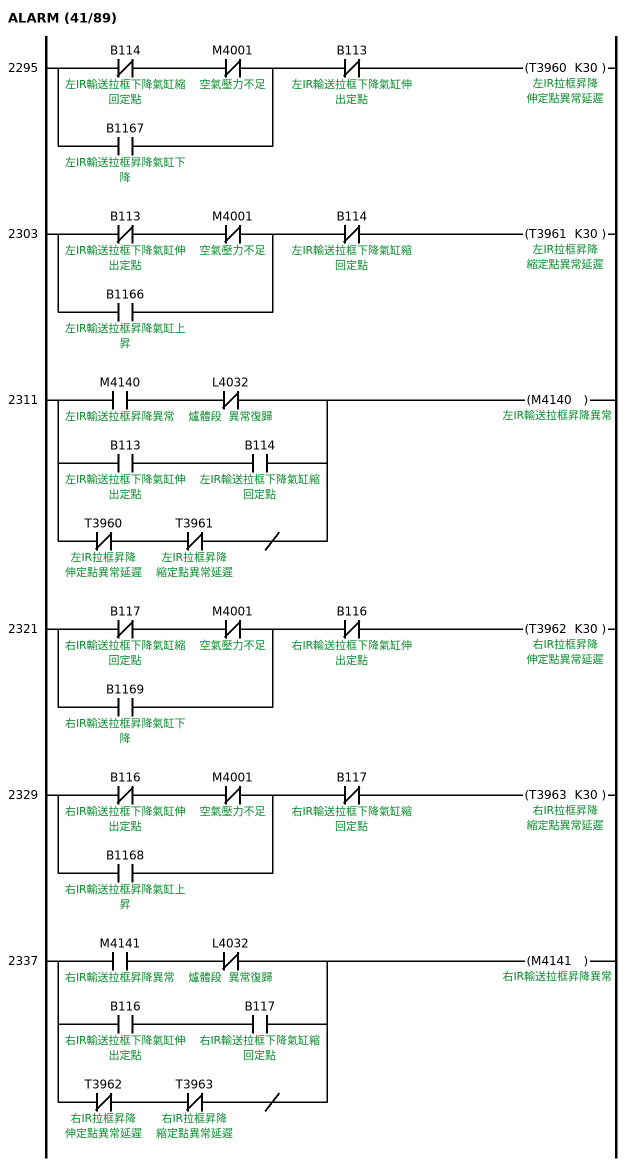
[picture p216: ladder of ALARM, rungs at steps 2295 to 2337]
2295  LDI     B114  ; 左IR輸送拉框下降氣缸縮回定點
      ANI     M4001  ; 空氣壓力不足
      OR      B1167  ; 左IR輸送拉框昇降氣缸下降
      ANI     B113  ; 左IR輸送拉框下降氣缸伸出定點
      OUT     T3960 K30  ; 左IR拉框昇降  伸定點異常延遲
2303  LDI     B113  ; 左IR輸送拉框下降氣缸伸出定點
      ANI     M4001  ; 空氣壓力不足
      OR      B1166  ; 左IR輸送拉框昇降氣缸上昇
      ANI     B114  ; 左IR輸送拉框下降氣缸縮回定點
      OUT     T3961 K30  ; 左IR拉框昇降  縮定點異常延遲
2311  LD      M4140  ; 左IR輸送拉框昇降異常
      ANI     L4032  ; 爐體段  異常復歸
      LD      B113  ; 左IR輸送拉框下降氣缸伸出定點
      AND     B114  ; 左IR輸送拉框下降氣缸縮回定點
      ORB
      LDI     T3960  ; 左IR拉框昇降  伸定點異常延遲
      ANI     T3961  ; 左IR拉框昇降  縮定點異常延遲
      INV
      ORB
      OUT     M4140  ; 左IR輸送拉框昇降異常
2321  LDI     B117  ; 右IR輸送拉框下降氣缸縮回定點
      ANI     M4001  ; 空氣壓力不足
      OR      B1169  ; 右IR輸送拉框昇降氣缸下降
      ANI     B116  ; 右IR輸送拉框下降氣缸伸出定點
      OUT     T3962 K30  ; 右IR拉框昇降  伸定點異常延遲
2329  LDI     B116  ; 右IR輸送拉框下降氣缸伸出定點
      ANI     M4001  ; 空氣壓力不足
      OR      B1168  ; 右IR輸送拉框昇降氣缸上昇
      ANI     B117  ; 右IR輸送拉框下降氣缸縮回定點
      OUT     T3963 K30  ; 右IR拉框昇降  縮定點異常延遲
2337  LD      M4141  ; 右IR輸送拉框昇降異常
      ANI     L4032  ; 爐體段  異常復歸
      LD      B116  ; 右IR輸送拉框下降氣缸伸出定點
      AND     B117  ; 右IR輸送拉框下降氣缸縮回定點
      ORB
      LDI     T3962  ; 右IR拉框昇降  伸定點異常延遲
      ANI     T3963  ; 右IR拉框昇降  縮定點異常延遲
      INV
      ORB
      OUT     M4141  ; 右IR輸送拉框昇降異常
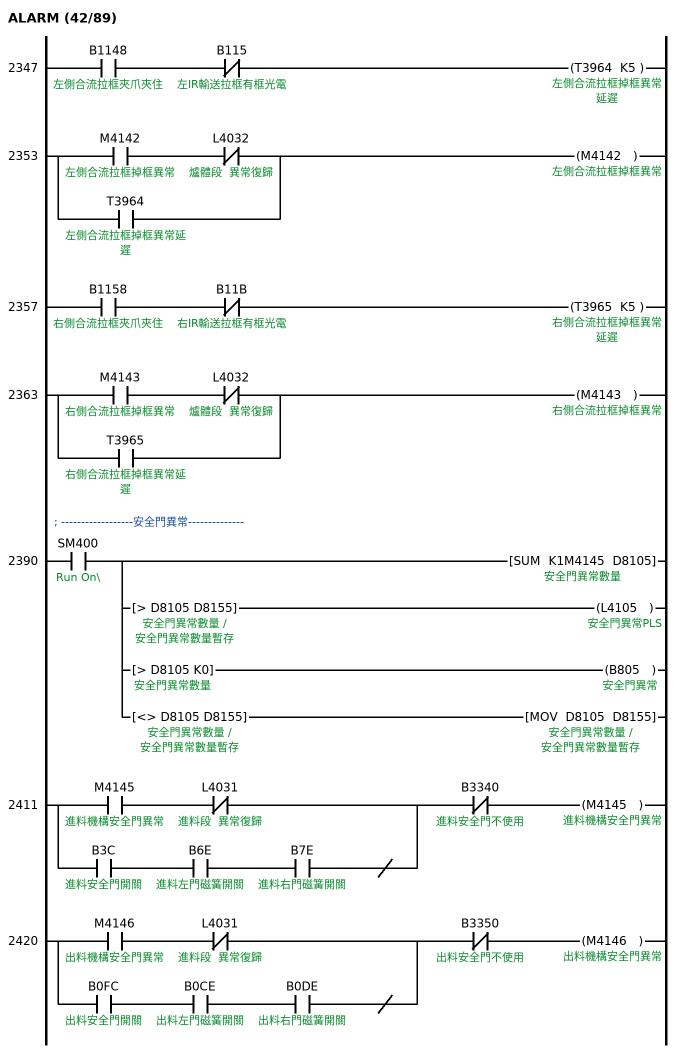
2347  LD      B1148  ; 左側合流拉框夾爪夾住
      ANI     B115  ; 左IR輸送拉框有框光電
      OUT     T3964 K5  ; 左側合流拉框掉框異常延遲
2353  LD      M4142  ; 左側合流拉框掉框異常
      ANI     L4032  ; 爐體段  異常復歸
      OR      T3964  ; 左側合流拉框掉框異常延遲
      OUT     M4142  ; 左側合流拉框掉框異常
2357  LD      B1158  ; 右側合流拉框夾爪夾住
      ANI     B11B  ; 右IR輸送拉框有框光電
      OUT     T3965 K5  ; 右側合流拉框掉框異常延遲
2363  LD      M4143  ; 右側合流拉框掉框異常
      ANI     L4032  ; 爐體段  異常復歸
      OR      T3965  ; 右側合流拉框掉框異常延遲
      OUT     M4143  ; 右側合流拉框掉框異常
; ------------------安全門異常--------------
2390  LD      SM400  ; Run On\
      SUM     K1M4145 D8105  ; 進料機構安全門異常 / 安全門異常數量
      MPS
      AND>    D8105 D8155  ; 安全門異常數量 / 安全門異常數量暫存
      OUT     L4105  ; 安全門異常PLS
      MRD
      AND>    D8105 K0  ; 安全門異常數量
      OUT     B805  ; 安全門異常
      MPP
      AND<>   D8105 D8155  ; 安全門異常數量 / 安全門異常數量暫存
      MOV     D8105 D8155
2411  LD      M4145  ; 進料機構安全門異常
      ANI     L4031  ; 進料段  異常復歸
      LD      B3C  ; 進料安全門開關
      AND     B6E  ; 進料左門磁簧開關
      AND     B7E  ; 進料右門磁簧開關
      INV
      ORB
      ANI     B3340  ; 進料安全門不使用
      OUT     M4145  ; 進料機構安全門異常
2420  LD      M4146  ; 出料機構安全門異常
      ANI     L4031  ; 進料段  異常復歸
      LD      B0FC  ; 出料安全門開關
      AND     B0CE  ; 出料左門磁簧開關
      AND     B0DE  ; 出料右門磁簧開關
      INV
      ORB
      ANI     B3350  ; 出料安全門不使用
      OUT     M4146  ; 出料機構安全門異常
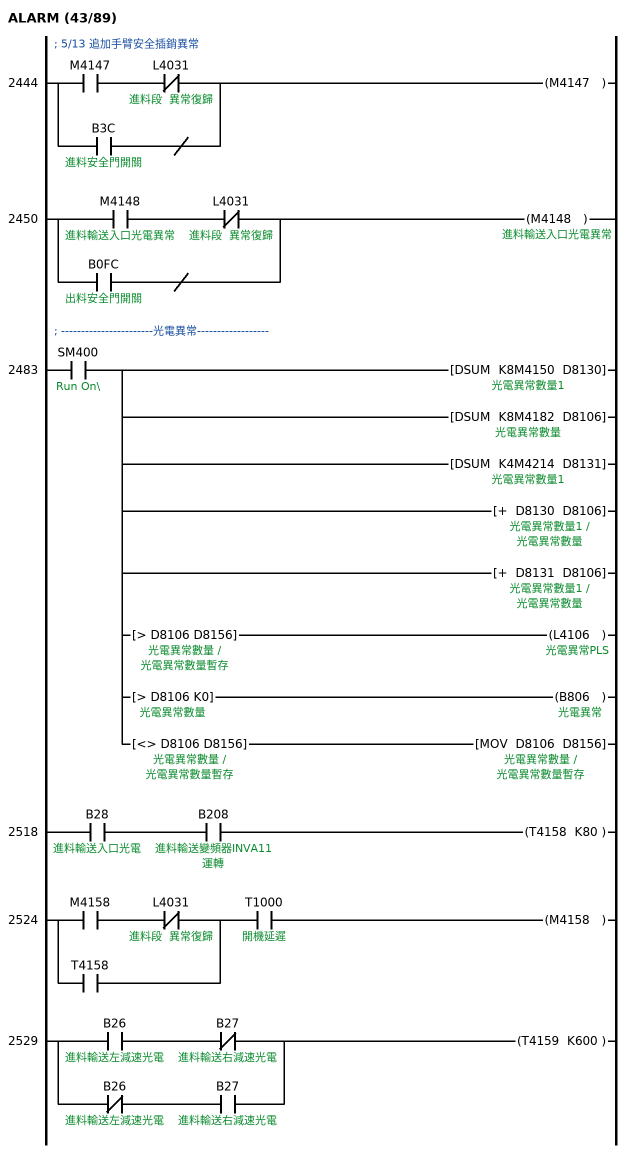
; 5/13 追加手臂安全插銷異常
2444  LD      M4147
      ANI     L4031  ; 進料段  異常復歸
      LD      B3C  ; 進料安全門開關
      INV
      ORB
      OUT     M4147
2450  LD      M4148  ; 進料輸送入口光電異常
      ANI     L4031  ; 進料段  異常復歸
      LD      B0FC  ; 出料安全門開關
      INV
      ORB
      OUT     M4148  ; 進料輸送入口光電異常
; -----------------------光電異常------------------
2483  LD      SM400  ; Run On\
      DSUM    K8M4150 D8130  ; 進料輸送有板光纖異常 / 光電異常數量1
      DSUM    K8M4182 D8106  ; 出料卡板異常 / 光電異常數量
      DSUM    K4M4214 D8131  ; 光電異常數量1
      +       D8130 D8106
      +       D8131 D8106
      MPS
      AND>    D8106 D8156  ; 光電異常數量 / 光電異常數量暫存
      OUT     L4106  ; 光電異常PLS
      MRD
      AND>    D8106 K0  ; 光電異常數量
      OUT     B806  ; 光電異常
      MPP
      AND<>   D8106 D8156  ; 光電異常數量 / 光電異常數量暫存
      MOV     D8106 D8156
2518  LD      B28  ; 進料輸送入口光電
      AND     B208  ; 進料輸送變頻器INVA11運轉
      OUT     T4158 K80
2524  LD      M4158
      ANI     L4031  ; 進料段  異常復歸
      OR      T4158
      AND     T1000  ; 開機延遲
      OUT     M4158
2529  LD      B26  ; 進料輸送左減速光電
      ANI     B27  ; 進料輸送右減速光電
      LDI     B26  ; 進料輸送左減速光電
      AND     B27  ; 進料輸送右減速光電
      ORB
      OUT     T4159 K600
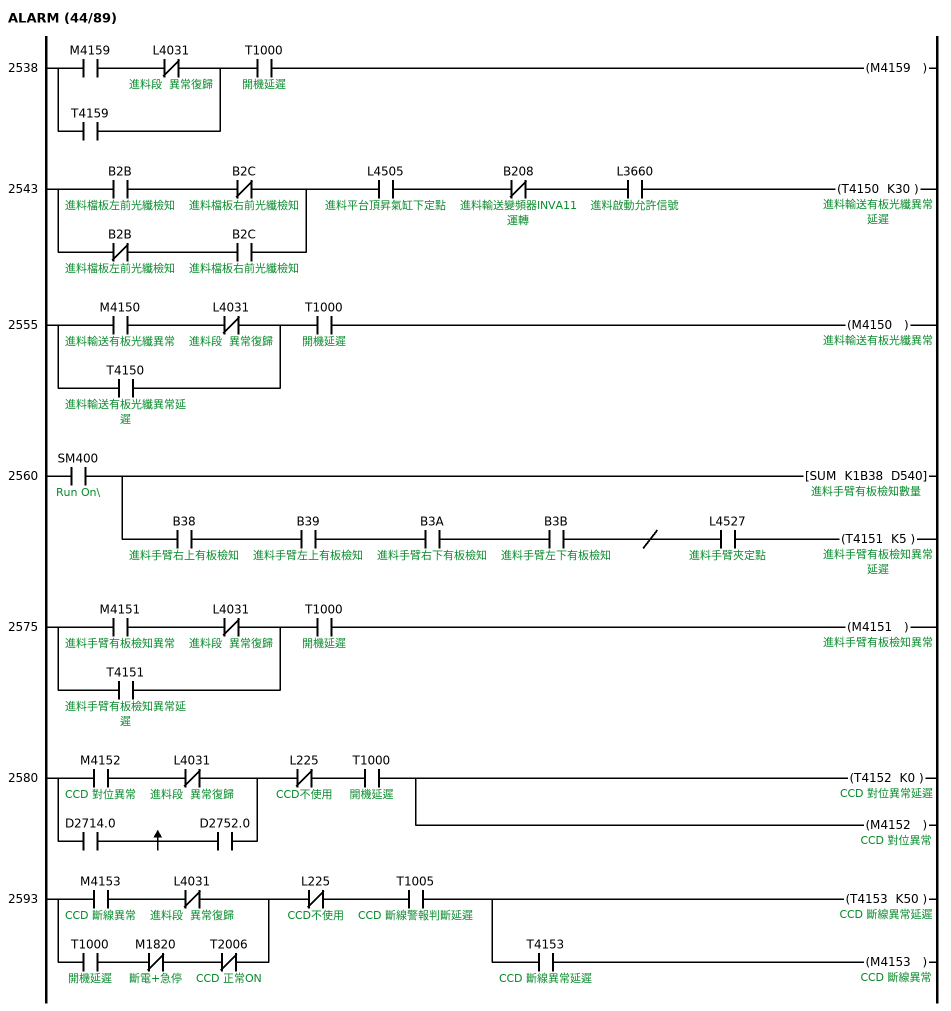
2538  LD      M4159
      ANI     L4031  ; 進料段  異常復歸
      OR      T4159
      AND     T1000  ; 開機延遲
      OUT     M4159
2543  LD      B2B  ; 進料檔板左前光纖檢知
      ANI     B2C  ; 進料檔板右前光纖檢知
      LDI     B2B  ; 進料檔板左前光纖檢知
      AND     B2C  ; 進料檔板右前光纖檢知
      ORB
      AND     L4505  ; 進料平台頂昇氣缸下定點
      ANI     B208  ; 進料輸送變頻器INVA11運轉
      AND     L3660  ; 進料啟動允許信號
      OUT     T4150 K30  ; 進料輸送有板光纖異常延遲
2555  LD      M4150  ; 進料輸送有板光纖異常
      ANI     L4031  ; 進料段  異常復歸
      OR      T4150  ; 進料輸送有板光纖異常延遲
      AND     T1000  ; 開機延遲
      OUT     M4150  ; 進料輸送有板光纖異常
2560  LD      SM400  ; Run On\
      SUM     K1B38 D540  ; 進料手臂右上有板檢知 / 進料手臂有板檢知數量
      AND     B38  ; 進料手臂右上有板檢知
      AND     B39  ; 進料手臂左上有板檢知
      AND     B3A  ; 進料手臂右下有板檢知
      AND     B3B  ; 進料手臂左下有板檢知
      INV
      AND     L4527  ; 進料手臂夾定點
      OUT     T4151 K5  ; 進料手臂有板檢知異常延遲
2575  LD      M4151  ; 進料手臂有板檢知異常
      ANI     L4031  ; 進料段  異常復歸
      OR      T4151  ; 進料手臂有板檢知異常延遲
      AND     T1000  ; 開機延遲
      OUT     M4151  ; 進料手臂有板檢知異常
2580  LD      M4152  ; CCD 對位異常
      ANI     L4031  ; 進料段  異常復歸
      LD      D2714.0
      MEP
      AND     D2752.0
      ORB
      ANI     L225  ; CCD不使用
      AND     T1000  ; 開機延遲
      OUT     T4152 K0  ; CCD 對位異常延遲
      OUT     M4152  ; CCD 對位異常
2593  LD      M4153  ; CCD 斷線異常
      ANI     L4031  ; 進料段  異常復歸
      LD      T1000  ; 開機延遲
      ANI     M1820  ; 斷電+急停
      ANI     T2006  ; CCD 正常ON
      ORB
      ANI     L225  ; CCD不使用
      AND     T1005  ; CCD 斷線警報判斷延遲
      OUT     T4153 K50  ; CCD 斷線異常延遲
      AND     T4153  ; CCD 斷線異常延遲
      OUT     M4153  ; CCD 斷線異常
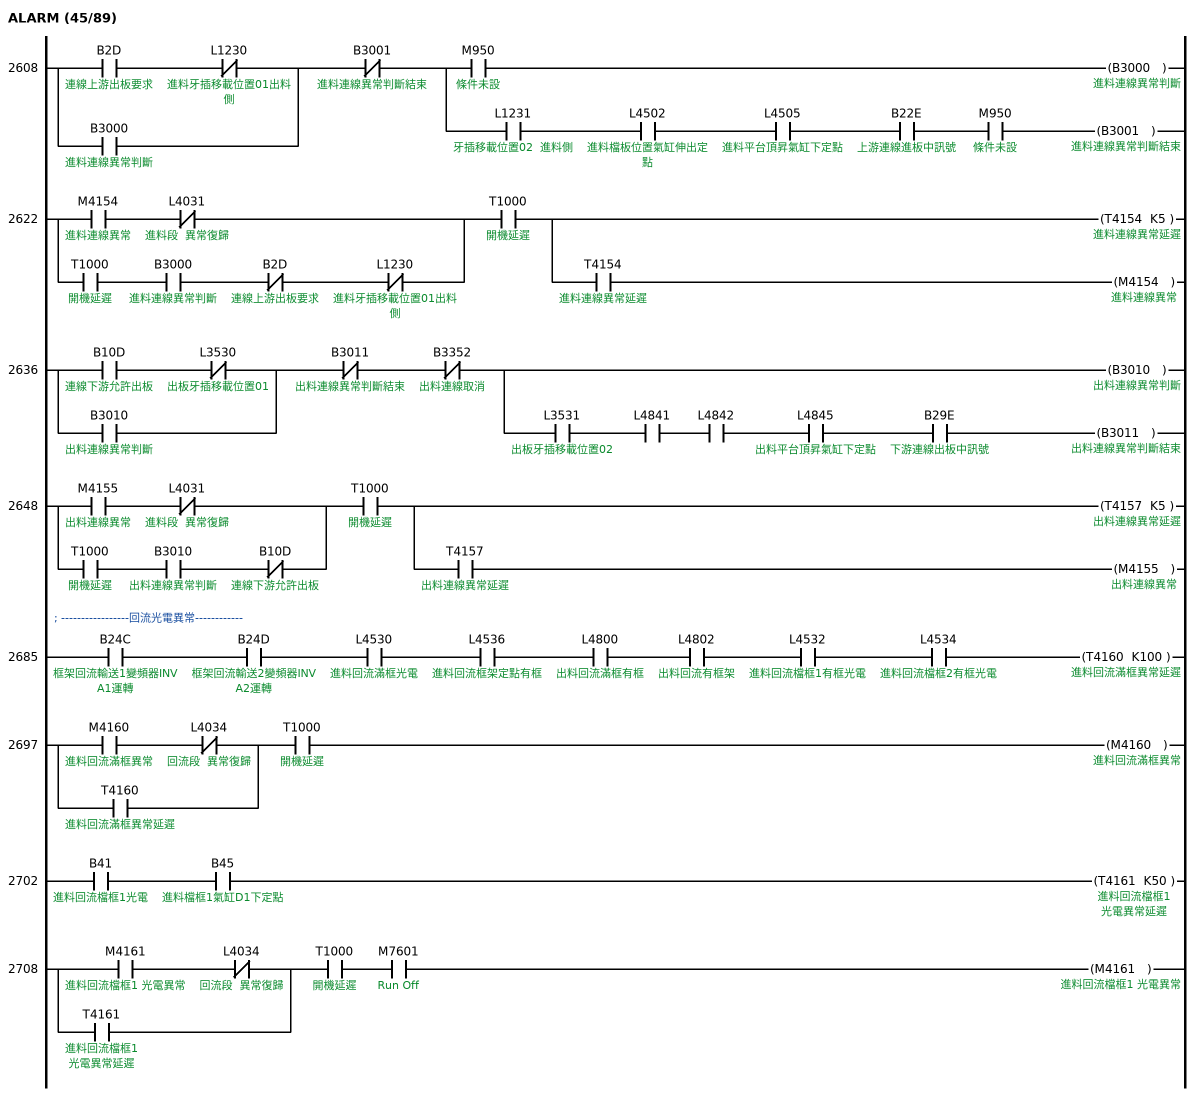
2608  LD      B2D  ; 連線上游出板要求
      ANI     L1230  ; 進料牙插移載位置01出料側
      OR      B3000  ; 進料連線異常判斷
      ANI     B3001  ; 進料連線異常判斷結束
      MPS
      AND     M950  ; 條件未設
      OUT     B3000  ; 進料連線異常判斷
      MPP
      AND     L1231  ; 牙插移載位置02  進料側
      AND     L4502  ; 進料檔板位置氣缸伸出定點
      AND     L4505  ; 進料平台頂昇氣缸下定點
      AND     B22E  ; 上游連線進板中訊號
      AND     M950  ; 條件未設
      OUT     B3001  ; 進料連線異常判斷結束
2622  LD      M4154  ; 進料連線異常
      ANI     L4031  ; 進料段  異常復歸
      LD      T1000  ; 開機延遲
      AND     B3000  ; 進料連線異常判斷
      ANI     B2D  ; 連線上游出板要求
      ANI     L1230  ; 進料牙插移載位置01出料側
      ORB
      AND     T1000  ; 開機延遲
      OUT     T4154 K5  ; 進料連線異常延遲
      AND     T4154  ; 進料連線異常延遲
      OUT     M4154  ; 進料連線異常
2636  LD      B10D  ; 連線下游允許出板
      ANI     L3530  ; 出板牙插移載位置01
      OR      B3010  ; 出料連線異常判斷
      ANI     B3011  ; 出料連線異常判斷結束
      ANI     B3352  ; 出料連線取消
      OUT     B3010  ; 出料連線異常判斷
      AND     L3531  ; 出板牙插移載位置02
      AND     L4841
      AND     L4842
      AND     L4845  ; 出料平台頂昇氣缸下定點
      AND     B29E  ; 下游連線出板中訊號
      OUT     B3011  ; 出料連線異常判斷結束
2648  LD      M4155  ; 出料連線異常
      ANI     L4031  ; 進料段  異常復歸
      LD      T1000  ; 開機延遲
      AND     B3010  ; 出料連線異常判斷
      ANI     B10D  ; 連線下游允許出板
      ORB
      AND     T1000  ; 開機延遲
      OUT     T4157 K5  ; 出料連線異常延遲
      AND     T4157  ; 出料連線異常延遲
      OUT     M4155  ; 出料連線異常
; -----------------回流光電異常------------
2685  LD      B24C  ; 框架回流輸送1變頻器INVA1運轉
      AND     B24D  ; 框架回流輸送2變頻器INVA2運轉
      AND     L4530  ; 進料回流滿框光電
      AND     L4536  ; 進料回流框架定點有框
      AND     L4800  ; 出料回流滿框有框
      AND     L4802  ; 出料回流有框架
      AND     L4532  ; 進料回流檔框1有框光電
      AND     L4534  ; 進料回流檔框2有框光電
      OUT     T4160 K100  ; 進料回流滿框異常延遲
2697  LD      M4160  ; 進料回流滿框異常
      ANI     L4034  ; 回流段  異常復歸
      OR      T4160  ; 進料回流滿框異常延遲
      AND     T1000  ; 開機延遲
      OUT     M4160  ; 進料回流滿框異常
2702  LD      B41  ; 進料回流檔框1光電
      AND     B45  ; 進料檔框1氣缸D1下定點
      OUT     T4161 K50  ; 進料回流檔框1 光電異常延遲
2708  LD      M4161  ; 進料回流檔框1 光電異常
      ANI     L4034  ; 回流段  異常復歸
      OR      T4161  ; 進料回流檔框1 光電異常延遲
      AND     T1000  ; 開機延遲
      AND     M7601  ; Run Off
      OUT     M4161  ; 進料回流檔框1 光電異常
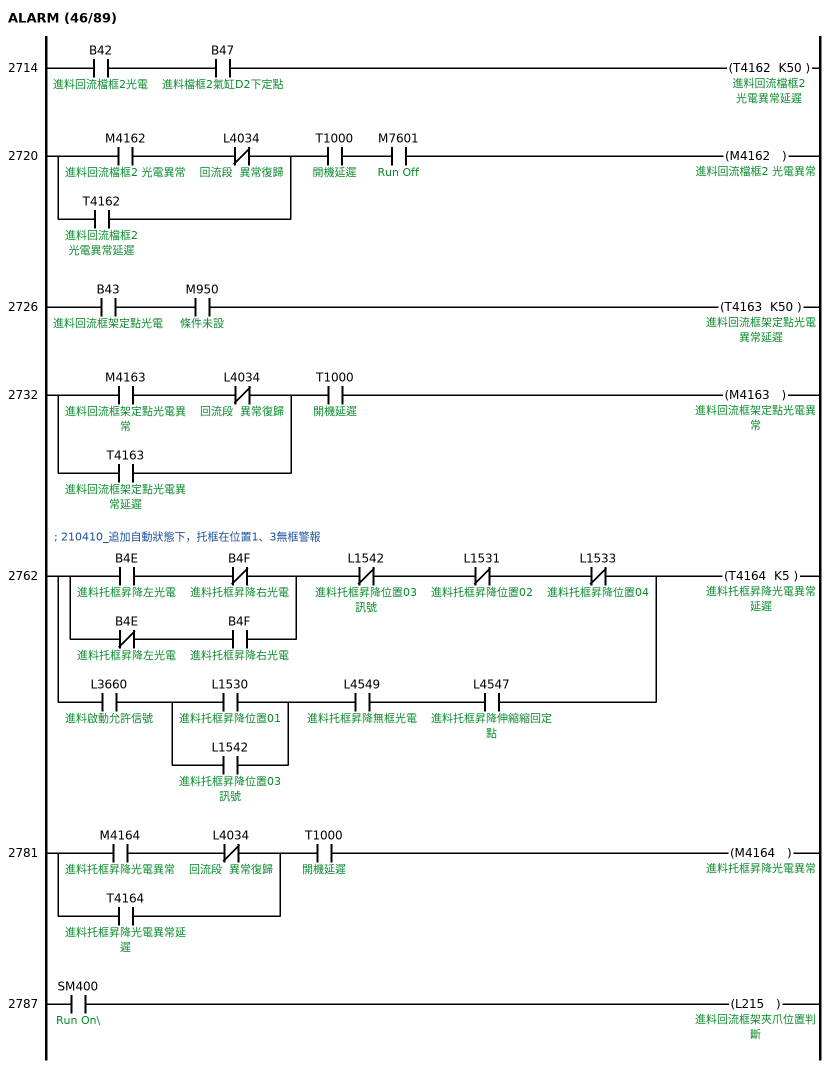
2714  LD      B42  ; 進料回流檔框2光電
      AND     B47  ; 進料檔框2氣缸D2下定點
      OUT     T4162 K50  ; 進料回流檔框2 光電異常延遲
2720  LD      M4162  ; 進料回流檔框2 光電異常
      ANI     L4034  ; 回流段  異常復歸
      OR      T4162  ; 進料回流檔框2 光電異常延遲
      AND     T1000  ; 開機延遲
      AND     M7601  ; Run Off
      OUT     M4162  ; 進料回流檔框2 光電異常
2726  LD      B43  ; 進料回流框架定點光電
      AND     M950  ; 條件未設
      OUT     T4163 K50  ; 進料回流框架定點光電異常延遲
2732  LD      M4163  ; 進料回流框架定點光電異常
      ANI     L4034  ; 回流段  異常復歸
      OR      T4163  ; 進料回流框架定點光電異常延遲
      AND     T1000  ; 開機延遲
      OUT     M4163  ; 進料回流框架定點光電異常
; 210410_追加自動狀態下，托框在位置1、3無框警報
2762  LD      B4E  ; 進料托框昇降左光電
      ANI     B4F  ; 進料托框昇降右光電
      LDI     B4E  ; 進料托框昇降左光電
      AND     B4F  ; 進料托框昇降右光電
      ORB
      ANI     L1542  ; 進料托框昇降位置03 訊號
      ANI     L1531  ; 進料托框昇降位置02
      ANI     L1533  ; 進料托框昇降位置04
      LD      L3660  ; 進料啟動允許信號
      LD      L1530  ; 進料托框昇降位置01
      OR      L1542  ; 進料托框昇降位置03 訊號
      ANB
      AND     L4549  ; 進料托框昇降無框光電
      AND     L4547  ; 進料托框昇降伸縮縮回定點
      ORB
      OUT     T4164 K5  ; 進料托框昇降光電異常延遲
2781  LD      M4164  ; 進料托框昇降光電異常
      ANI     L4034  ; 回流段  異常復歸
      OR      T4164  ; 進料托框昇降光電異常延遲
      AND     T1000  ; 開機延遲
      OUT     M4164  ; 進料托框昇降光電異常
2787  LD      SM400  ; Run On\
      OUT     L215  ; 進料回流框架夾爪位置判斷
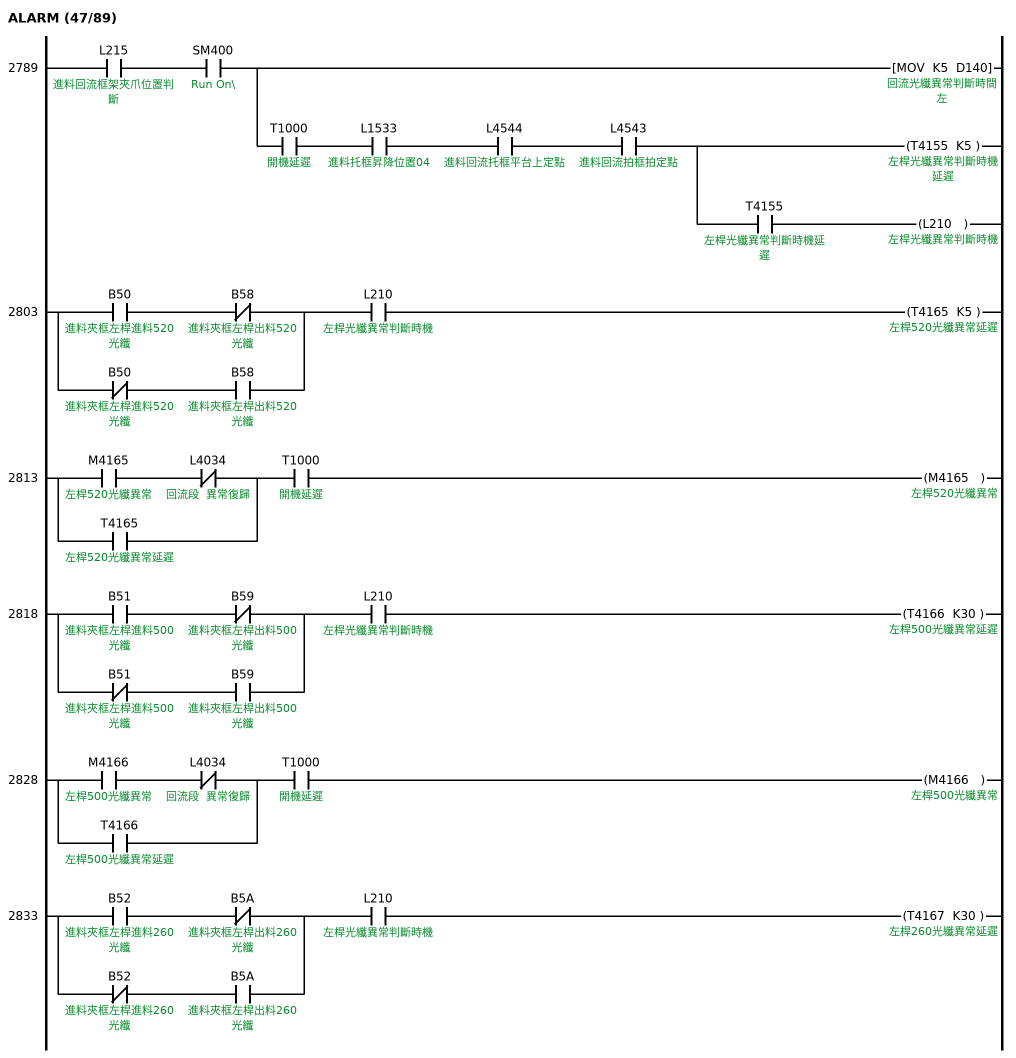
2789  LD      L215  ; 進料回流框架夾爪位置判斷
      AND     SM400  ; Run On\
      MOV     K5 D140  ; 回流光纖異常判斷時間左
      AND     T1000  ; 開機延遲
      AND     L1533  ; 進料托框昇降位置04
      AND     L4544  ; 進料回流托框平台上定點
      AND     L4543  ; 進料回流拍框拍定點
      OUT     T4155 K5  ; 左桿光纖異常判斷時機延遲
      AND     T4155  ; 左桿光纖異常判斷時機延遲
      OUT     L210  ; 左桿光纖異常判斷時機
2803  LD      B50  ; 進料夾框左桿進料520 光纖
      ANI     B58  ; 進料夾框左桿出料520 光纖
      LDI     B50  ; 進料夾框左桿進料520 光纖
      AND     B58  ; 進料夾框左桿出料520 光纖
      ORB
      AND     L210  ; 左桿光纖異常判斷時機
      OUT     T4165 K5  ; 左桿520光纖異常延遲
2813  LD      M4165  ; 左桿520光纖異常
      ANI     L4034  ; 回流段  異常復歸
      OR      T4165  ; 左桿520光纖異常延遲
      AND     T1000  ; 開機延遲
      OUT     M4165  ; 左桿520光纖異常
2818  LD      B51  ; 進料夾框左桿進料500 光纖
      ANI     B59  ; 進料夾框左桿出料500 光纖
      LDI     B51  ; 進料夾框左桿進料500 光纖
      AND     B59  ; 進料夾框左桿出料500 光纖
      ORB
      AND     L210  ; 左桿光纖異常判斷時機
      OUT     T4166 K30  ; 左桿500光纖異常延遲
2828  LD      M4166  ; 左桿500光纖異常
      ANI     L4034  ; 回流段  異常復歸
      OR      T4166  ; 左桿500光纖異常延遲
      AND     T1000  ; 開機延遲
      OUT     M4166  ; 左桿500光纖異常
2833  LD      B52  ; 進料夾框左桿進料260 光纖
      ANI     B5A  ; 進料夾框左桿出料260 光纖
      LDI     B52  ; 進料夾框左桿進料260 光纖
      AND     B5A  ; 進料夾框左桿出料260 光纖
      ORB
      AND     L210  ; 左桿光纖異常判斷時機
      OUT     T4167 K30  ; 左桿260光纖異常延遲
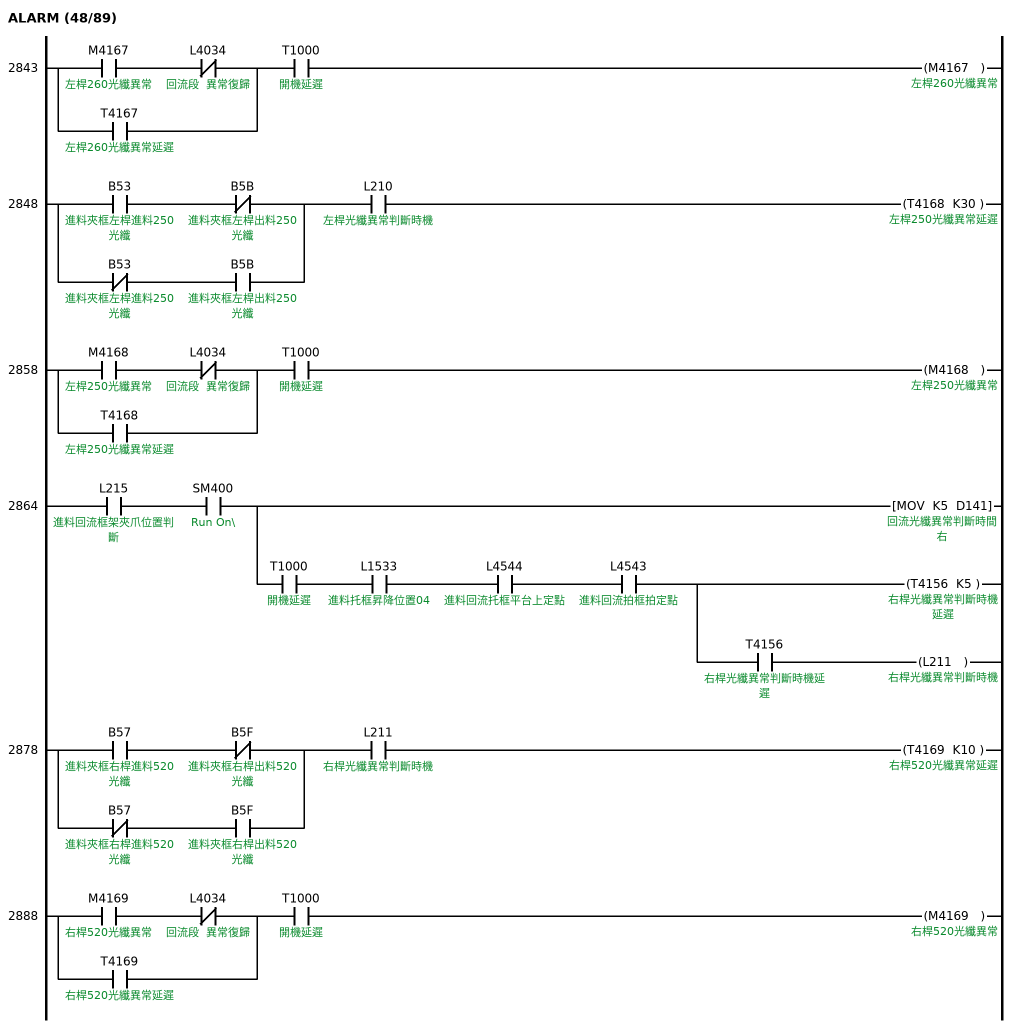
2843  LD      M4167  ; 左桿260光纖異常
      ANI     L4034  ; 回流段  異常復歸
      OR      T4167  ; 左桿260光纖異常延遲
      AND     T1000  ; 開機延遲
      OUT     M4167  ; 左桿260光纖異常
2848  LD      B53  ; 進料夾框左桿進料250 光纖
      ANI     B5B  ; 進料夾框左桿出料250 光纖
      LDI     B53  ; 進料夾框左桿進料250 光纖
      AND     B5B  ; 進料夾框左桿出料250 光纖
      ORB
      AND     L210  ; 左桿光纖異常判斷時機
      OUT     T4168 K30  ; 左桿250光纖異常延遲
2858  LD      M4168  ; 左桿250光纖異常
      ANI     L4034  ; 回流段  異常復歸
      OR      T4168  ; 左桿250光纖異常延遲
      AND     T1000  ; 開機延遲
      OUT     M4168  ; 左桿250光纖異常
2864  LD      L215  ; 進料回流框架夾爪位置判斷
      AND     SM400  ; Run On\
      MOV     K5 D141  ; 回流光纖異常判斷時間右
      AND     T1000  ; 開機延遲
      AND     L1533  ; 進料托框昇降位置04
      AND     L4544  ; 進料回流托框平台上定點
      AND     L4543  ; 進料回流拍框拍定點
      OUT     T4156 K5  ; 右桿光纖異常判斷時機延遲
      AND     T4156  ; 右桿光纖異常判斷時機延遲
      OUT     L211  ; 右桿光纖異常判斷時機
2878  LD      B57  ; 進料夾框右桿進料520 光纖
      ANI     B5F  ; 進料夾框右桿出料520 光纖
      LDI     B57  ; 進料夾框右桿進料520 光纖
      AND     B5F  ; 進料夾框右桿出料520 光纖
      ORB
      AND     L211  ; 右桿光纖異常判斷時機
      OUT     T4169 K10  ; 右桿520光纖異常延遲
2888  LD      M4169  ; 右桿520光纖異常
      ANI     L4034  ; 回流段  異常復歸
      OR      T4169  ; 右桿520光纖異常延遲
      AND     T1000  ; 開機延遲
      OUT     M4169  ; 右桿520光纖異常
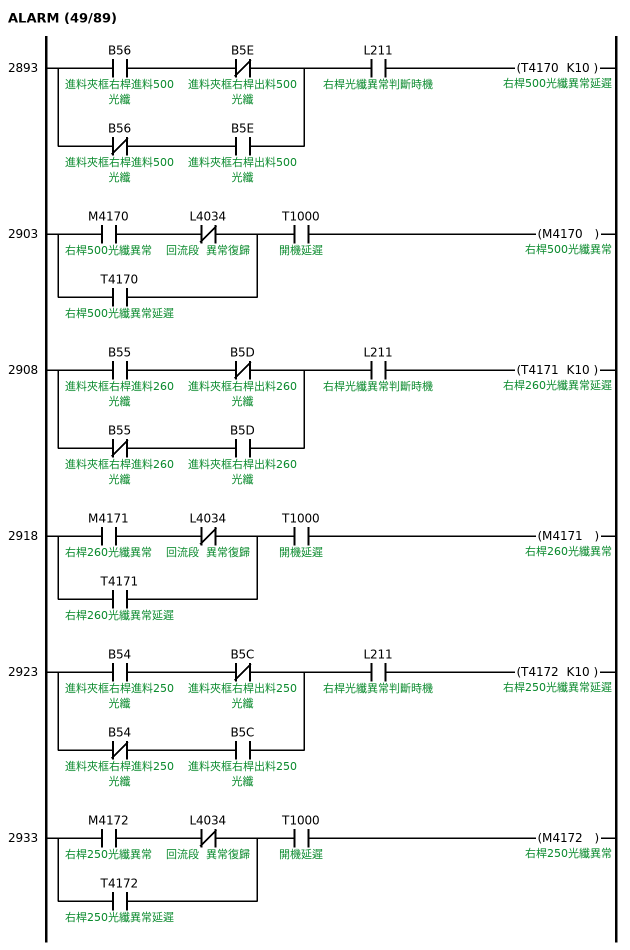
2893  LD      B56  ; 進料夾框右桿進料500 光纖
      ANI     B5E  ; 進料夾框右桿出料500 光纖
      LDI     B56  ; 進料夾框右桿進料500 光纖
      AND     B5E  ; 進料夾框右桿出料500 光纖
      ORB
      AND     L211  ; 右桿光纖異常判斷時機
      OUT     T4170 K10  ; 右桿500光纖異常延遲
2903  LD      M4170  ; 右桿500光纖異常
      ANI     L4034  ; 回流段  異常復歸
      OR      T4170  ; 右桿500光纖異常延遲
      AND     T1000  ; 開機延遲
      OUT     M4170  ; 右桿500光纖異常
2908  LD      B55  ; 進料夾框右桿進料260 光纖
      ANI     B5D  ; 進料夾框右桿出料260 光纖
      LDI     B55  ; 進料夾框右桿進料260 光纖
      AND     B5D  ; 進料夾框右桿出料260 光纖
      ORB
      AND     L211  ; 右桿光纖異常判斷時機
      OUT     T4171 K10  ; 右桿260光纖異常延遲
2918  LD      M4171  ; 右桿260光纖異常
      ANI     L4034  ; 回流段  異常復歸
      OR      T4171  ; 右桿260光纖異常延遲
      AND     T1000  ; 開機延遲
      OUT     M4171  ; 右桿260光纖異常
2923  LD      B54  ; 進料夾框右桿進料250 光纖
      ANI     B5C  ; 進料夾框右桿出料250 光纖
      LDI     B54  ; 進料夾框右桿進料250 光纖
      AND     B5C  ; 進料夾框右桿出料250 光纖
      ORB
      AND     L211  ; 右桿光纖異常判斷時機
      OUT     T4172 K10  ; 右桿250光纖異常延遲
2933  LD      M4172  ; 右桿250光纖異常
      ANI     L4034  ; 回流段  異常復歸
      OR      T4172  ; 右桿250光纖異常延遲
      AND     T1000  ; 開機延遲
      OUT     M4172  ; 右桿250光纖異常
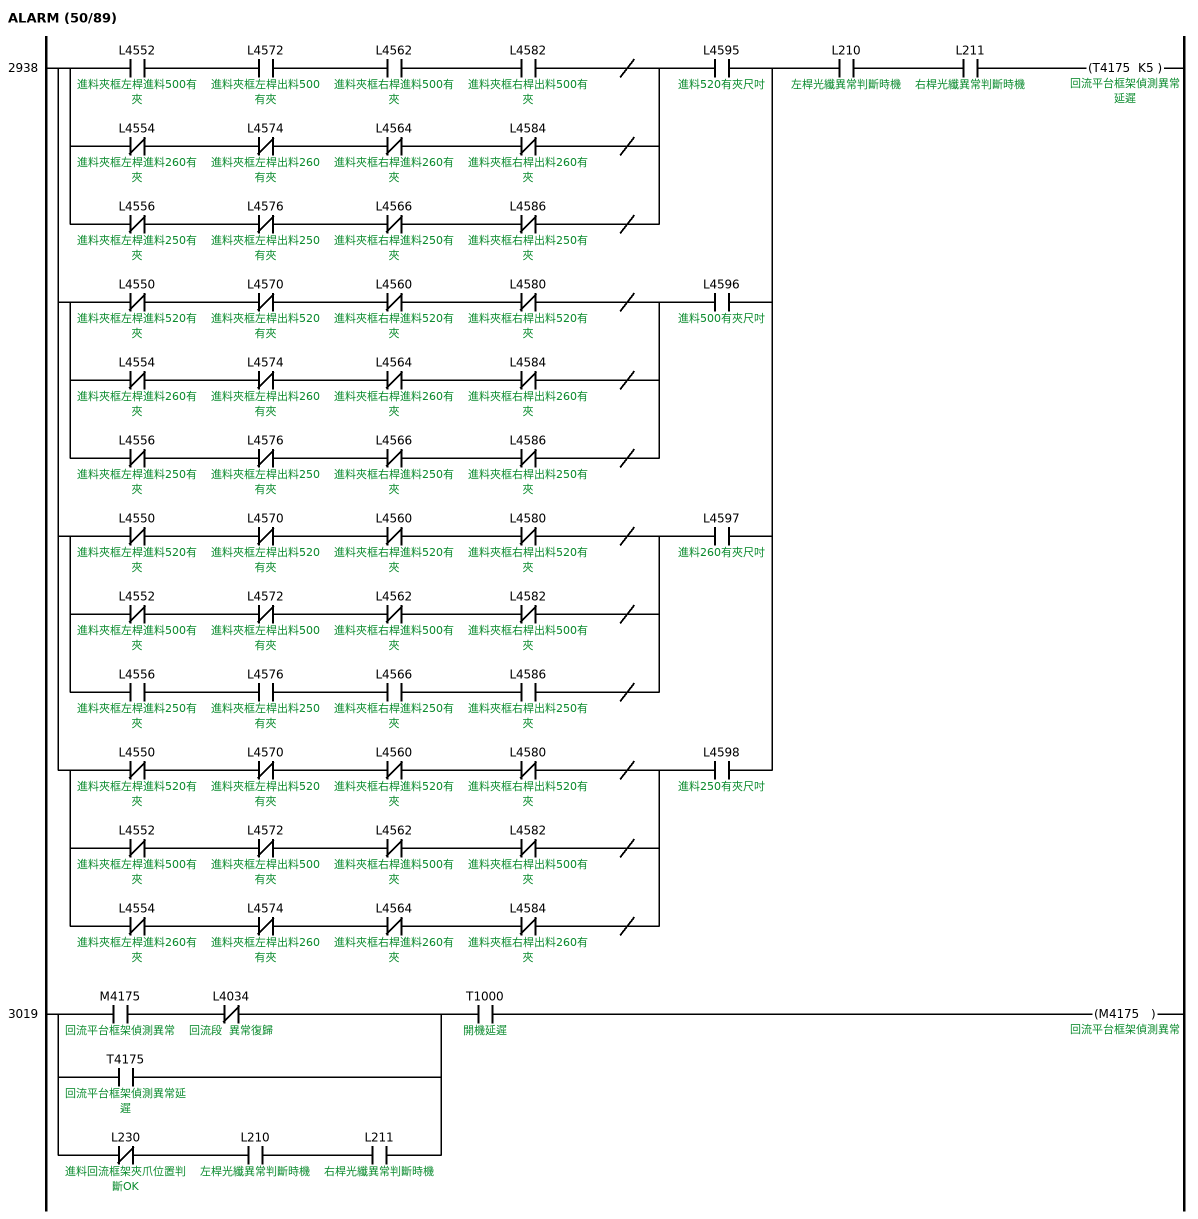
2938  LD      L4552  ; 進料夾框左桿進料500有夾
      AND     L4572  ; 進料夾框左桿出料500 有夾
      AND     L4562  ; 進料夾框右桿進料500有夾
      AND     L4582  ; 進料夾框右桿出料500有夾
      INV
      LDI     L4554  ; 進料夾框左桿進料260有夾
      ANI     L4574  ; 進料夾框左桿出料260 有夾
      ANI     L4564  ; 進料夾框右桿進料260有夾
      ANI     L4584  ; 進料夾框右桿出料260有夾
      INV
      ORB
      LDI     L4556  ; 進料夾框左桿進料250有夾
      ANI     L4576  ; 進料夾框左桿出料250 有夾
      ANI     L4566  ; 進料夾框右桿進料250有夾
      ANI     L4586  ; 進料夾框右桿出料250有夾
      INV
      ORB
      AND     L4595  ; 進料520有夾尺吋
      LDI     L4550  ; 進料夾框左桿進料520有夾
      ANI     L4570  ; 進料夾框左桿出料520 有夾
      ANI     L4560  ; 進料夾框右桿進料520有夾
      ANI     L4580  ; 進料夾框右桿出料520有夾
      INV
      LDI     L4554  ; 進料夾框左桿進料260有夾
      ANI     L4574  ; 進料夾框左桿出料260 有夾
      ANI     L4564  ; 進料夾框右桿進料260有夾
      ANI     L4584  ; 進料夾框右桿出料260有夾
      INV
      ORB
      LDI     L4556  ; 進料夾框左桿進料250有夾
      ANI     L4576  ; 進料夾框左桿出料250 有夾
      ANI     L4566  ; 進料夾框右桿進料250有夾
      ANI     L4586  ; 進料夾框右桿出料250有夾
      INV
      ORB
      AND     L4596  ; 進料500有夾尺吋
      ORB
      LDI     L4550  ; 進料夾框左桿進料520有夾
      ANI     L4570  ; 進料夾框左桿出料520 有夾
      ANI     L4560  ; 進料夾框右桿進料520有夾
      ANI     L4580  ; 進料夾框右桿出料520有夾
      INV
      LDI     L4552  ; 進料夾框左桿進料500有夾
      ANI     L4572  ; 進料夾框左桿出料500 有夾
      ANI     L4562  ; 進料夾框右桿進料500有夾
      ANI     L4582  ; 進料夾框右桿出料500有夾
      INV
      ORB
      LD      L4556  ; 進料夾框左桿進料250有夾
      AND     L4576  ; 進料夾框左桿出料250 有夾
      AND     L4566  ; 進料夾框右桿進料250有夾
      AND     L4586  ; 進料夾框右桿出料250有夾
      INV
      ORB
      AND     L4597  ; 進料260有夾尺吋
      ORB
      LDI     L4550  ; 進料夾框左桿進料520有夾
      ANI     L4570  ; 進料夾框左桿出料520 有夾
      ANI     L4560  ; 進料夾框右桿進料520有夾
      ANI     L4580  ; 進料夾框右桿出料520有夾
      INV
      LDI     L4552  ; 進料夾框左桿進料500有夾
      ANI     L4572  ; 進料夾框左桿出料500 有夾
      ANI     L4562  ; 進料夾框右桿進料500有夾
      ANI     L4582  ; 進料夾框右桿出料500有夾
      INV
      ORB
      LDI     L4554  ; 進料夾框左桿進料260有夾
      ANI     L4574  ; 進料夾框左桿出料260 有夾
      ANI     L4564  ; 進料夾框右桿進料260有夾
      ANI     L4584  ; 進料夾框右桿出料260有夾
      INV
      ORB
      AND     L4598  ; 進料250有夾尺吋
      ORB
      AND     L210  ; 左桿光纖異常判斷時機
      AND     L211  ; 右桿光纖異常判斷時機
      OUT     T4175 K5  ; 回流平台框架偵測異常延遲
3019  LD      M4175  ; 回流平台框架偵測異常
      ANI     L4034  ; 回流段  異常復歸
      OR      T4175  ; 回流平台框架偵測異常延遲
      LDI     L230  ; 進料回流框架夾爪位置判斷OK
      AND     L210  ; 左桿光纖異常判斷時機
      AND     L211  ; 右桿光纖異常判斷時機
      ORB
      AND     T1000  ; 開機延遲
      OUT     M4175  ; 回流平台框架偵測異常
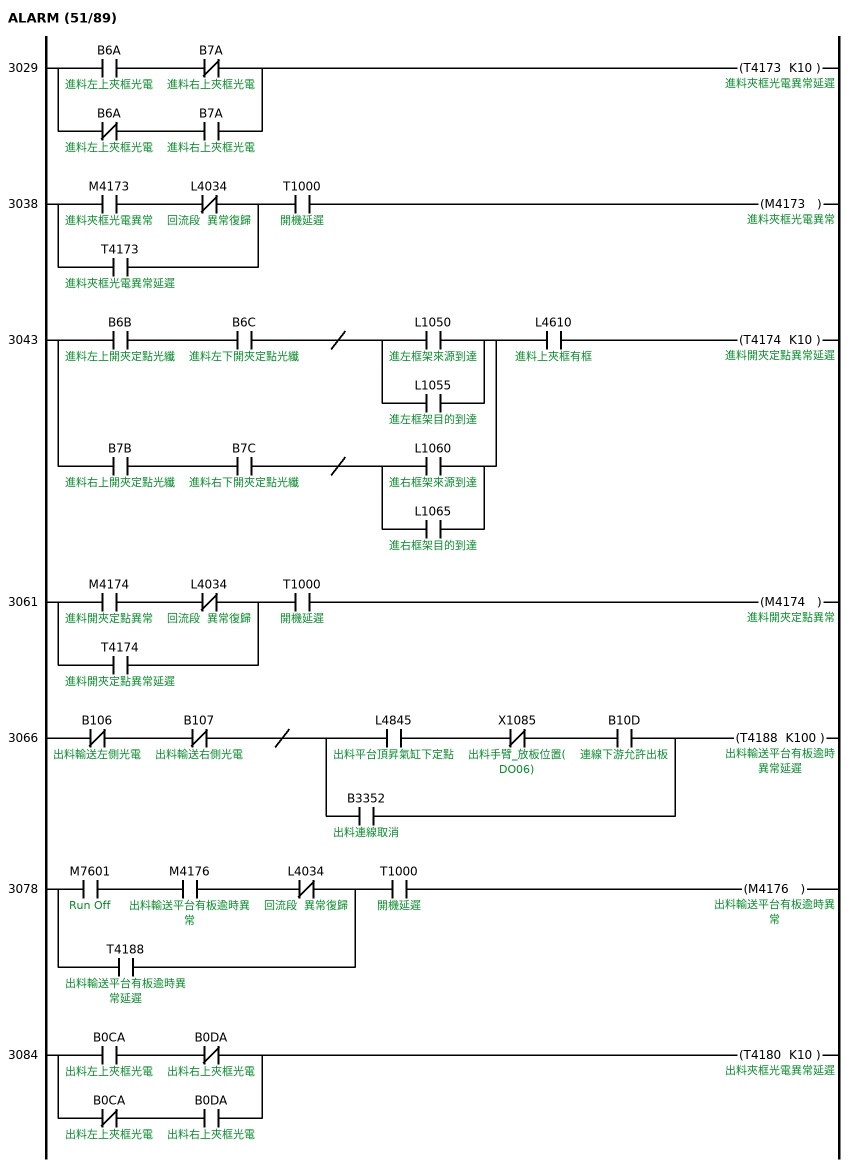
3029  LD      B6A  ; 進料左上夾框光電
      ANI     B7A  ; 進料右上夾框光電
      LDI     B6A  ; 進料左上夾框光電
      AND     B7A  ; 進料右上夾框光電
      ORB
      OUT     T4173 K10  ; 進料夾框光電異常延遲
3038  LD      M4173  ; 進料夾框光電異常
      ANI     L4034  ; 回流段  異常復歸
      OR      T4173  ; 進料夾框光電異常延遲
      AND     T1000  ; 開機延遲
      OUT     M4173  ; 進料夾框光電異常
3043  LD      B6B  ; 進料左上開夾定點光纖
      AND     B6C  ; 進料左下開夾定點光纖
      INV
      LD      L1050  ; 進左框架來源到達
      OR      L1055  ; 進左框架目的到達
      ANB
      LD      B7B  ; 進料右上開夾定點光纖
      AND     B7C  ; 進料右下開夾定點光纖
      INV
      LD      L1060  ; 進右框架來源到達
      OR      L1065  ; 進右框架目的到達
      ANB
      ORB
      AND     L4610  ; 進料上夾框有框
      OUT     T4174 K10  ; 進料開夾定點異常延遲
3061  LD      M4174  ; 進料開夾定點異常
      ANI     L4034  ; 回流段  異常復歸
      OR      T4174  ; 進料開夾定點異常延遲
      AND     T1000  ; 開機延遲
      OUT     M4174  ; 進料開夾定點異常
3066  LDI     B106  ; 出料輸送左側光電
      ANI     B107  ; 出料輸送右側光電
      INV
      LD      L4845  ; 出料平台頂昇氣缸下定點
      ANI     X1085  ; 出料手臂_放板位置(DO06)
      AND     B10D  ; 連線下游允許出板
      OR      B3352  ; 出料連線取消
      ANB
      OUT     T4188 K100  ; 出料輸送平台有板逾時異常延遲
3078  LD      M7601  ; Run Off
      AND     M4176  ; 出料輸送平台有板逾時異常
      ANI     L4034  ; 回流段  異常復歸
      OR      T4188  ; 出料輸送平台有板逾時異常延遲
      AND     T1000  ; 開機延遲
      OUT     M4176  ; 出料輸送平台有板逾時異常
3084  LD      B0CA  ; 出料左上夾框光電
      ANI     B0DA  ; 出料右上夾框光電
      LDI     B0CA  ; 出料左上夾框光電
      AND     B0DA  ; 出料右上夾框光電
      ORB
      OUT     T4180 K10  ; 出料夾框光電異常延遲
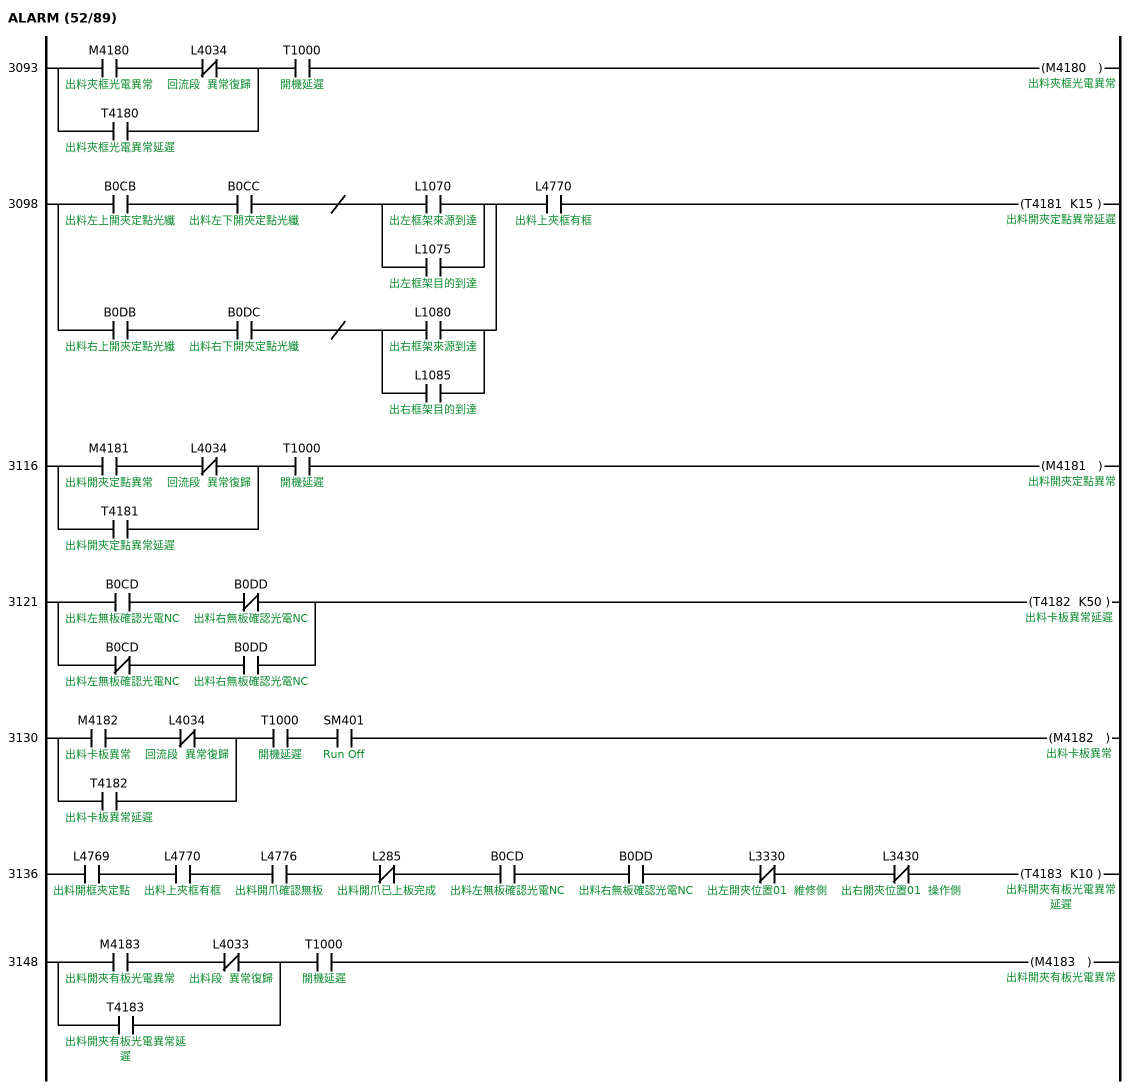
3093  LD      M4180  ; 出料夾框光電異常
      ANI     L4034  ; 回流段  異常復歸
      OR      T4180  ; 出料夾框光電異常延遲
      AND     T1000  ; 開機延遲
      OUT     M4180  ; 出料夾框光電異常
3098  LD      B0CB  ; 出料左上開夾定點光纖
      AND     B0CC  ; 出料左下開夾定點光纖
      INV
      LD      L1070  ; 出左框架來源到達
      OR      L1075  ; 出左框架目的到達
      ANB
      LD      B0DB  ; 出料右上開夾定點光纖
      AND     B0DC  ; 出料右下開夾定點光纖
      INV
      LD      L1080  ; 出右框架來源到達
      OR      L1085  ; 出右框架目的到達
      ANB
      ORB
      AND     L4770  ; 出料上夾框有框
      OUT     T4181 K15  ; 出料開夾定點異常延遲
3116  LD      M4181  ; 出料開夾定點異常
      ANI     L4034  ; 回流段  異常復歸
      OR      T4181  ; 出料開夾定點異常延遲
      AND     T1000  ; 開機延遲
      OUT     M4181  ; 出料開夾定點異常
3121  LD      B0CD  ; 出料左無板確認光電NC
      ANI     B0DD  ; 出料右無板確認光電NC
      LDI     B0CD  ; 出料左無板確認光電NC
      AND     B0DD  ; 出料右無板確認光電NC
      ORB
      OUT     T4182 K50  ; 出料卡板異常延遲
3130  LD      M4182  ; 出料卡板異常
      ANI     L4034  ; 回流段  異常復歸
      OR      T4182  ; 出料卡板異常延遲
      AND     T1000  ; 開機延遲
      AND     SM401  ; Run Off
      OUT     M4182  ; 出料卡板異常
3136  LD      L4769  ; 出料開框夾定點
      AND     L4770  ; 出料上夾框有框
      AND     L4776  ; 出料開爪確認無板
      ANI     L285  ; 出料開爪已上板完成
      AND     B0CD  ; 出料左無板確認光電NC
      AND     B0DD  ; 出料右無板確認光電NC
      ANI     L3330  ; 出左開夾位置01  維修側
      ANI     L3430  ; 出右開夾位置01  操作側
      OUT     T4183 K10  ; 出料開夾有板光電異常延遲
3148  LD      M4183  ; 出料開夾有板光電異常
      ANI     L4033  ; 出料段  異常復歸
      OR      T4183  ; 出料開夾有板光電異常延遲
      AND     T1000  ; 開機延遲
      OUT     M4183  ; 出料開夾有板光電異常
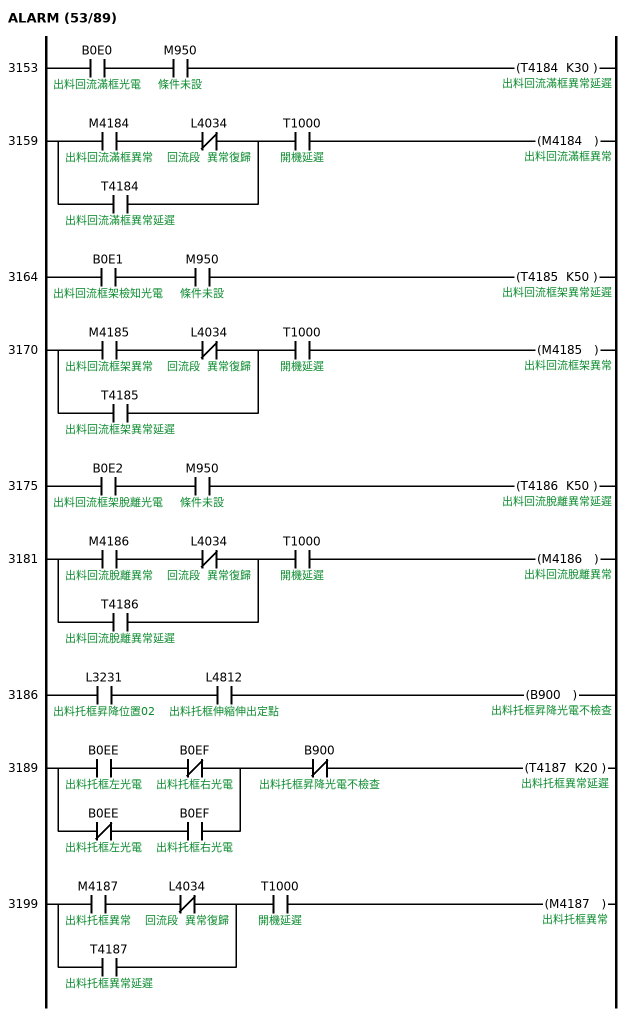
3153  LD      B0E0  ; 出料回流滿框光電
      AND     M950  ; 條件未設
      OUT     T4184 K30  ; 出料回流滿框異常延遲
3159  LD      M4184  ; 出料回流滿框異常
      ANI     L4034  ; 回流段  異常復歸
      OR      T4184  ; 出料回流滿框異常延遲
      AND     T1000  ; 開機延遲
      OUT     M4184  ; 出料回流滿框異常
3164  LD      B0E1  ; 出料回流框架檢知光電
      AND     M950  ; 條件未設
      OUT     T4185 K50  ; 出料回流框架異常延遲
3170  LD      M4185  ; 出料回流框架異常
      ANI     L4034  ; 回流段  異常復歸
      OR      T4185  ; 出料回流框架異常延遲
      AND     T1000  ; 開機延遲
      OUT     M4185  ; 出料回流框架異常
3175  LD      B0E2  ; 出料回流框架脫離光電
      AND     M950  ; 條件未設
      OUT     T4186 K50  ; 出料回流脫離異常延遲
3181  LD      M4186  ; 出料回流脫離異常
      ANI     L4034  ; 回流段  異常復歸
      OR      T4186  ; 出料回流脫離異常延遲
      AND     T1000  ; 開機延遲
      OUT     M4186  ; 出料回流脫離異常
3186  LD      L3231  ; 出料托框昇降位置02
      AND     L4812  ; 出料托框伸縮伸出定點
      OUT     B900  ; 出料托框昇降光電不檢查
3189  LD      B0EE  ; 出料托框左光電
      ANI     B0EF  ; 出料托框右光電
      LDI     B0EE  ; 出料托框左光電
      AND     B0EF  ; 出料托框右光電
      ORB
      ANI     B900  ; 出料托框昇降光電不檢查
      OUT     T4187 K20  ; 出料托框異常延遲
3199  LD      M4187  ; 出料托框異常
      ANI     L4034  ; 回流段  異常復歸
      OR      T4187  ; 出料托框異常延遲
      AND     T1000  ; 開機延遲
      OUT     M4187  ; 出料托框異常
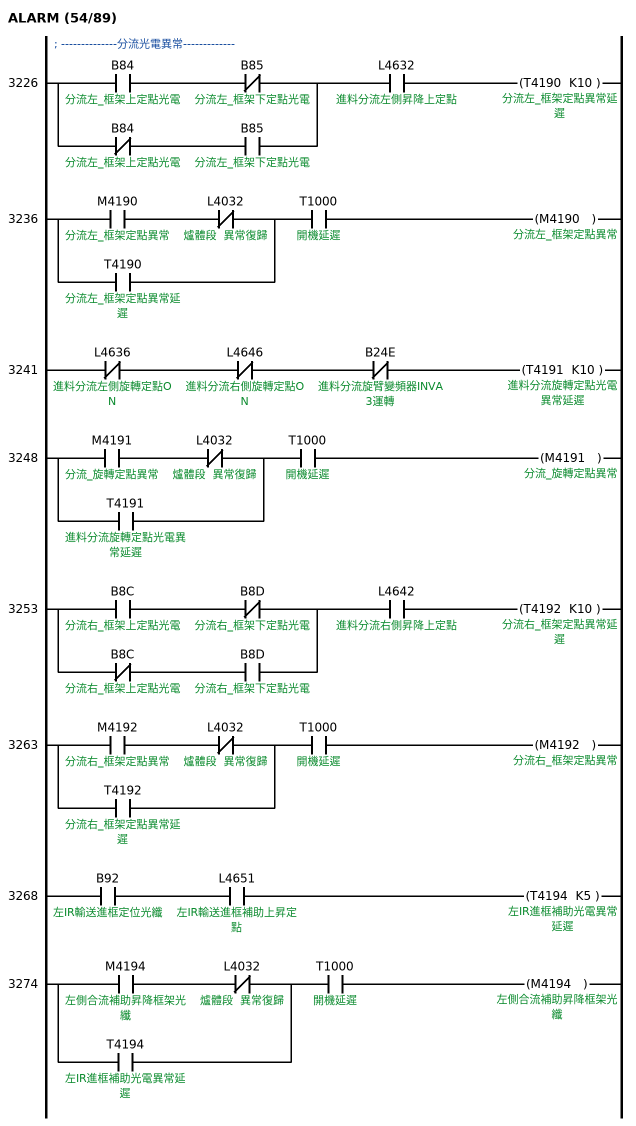
; --------------分流光電異常-------------
3226  LD      B84  ; 分流左_框架上定點光電
      ANI     B85  ; 分流左_框架下定點光電
      LDI     B84  ; 分流左_框架上定點光電
      AND     B85  ; 分流左_框架下定點光電
      ORB
      AND     L4632  ; 進料分流左側昇降上定點
      OUT     T4190 K10  ; 分流左_框架定點異常延遲
3236  LD      M4190  ; 分流左_框架定點異常
      ANI     L4032  ; 爐體段  異常復歸
      OR      T4190  ; 分流左_框架定點異常延遲
      AND     T1000  ; 開機延遲
      OUT     M4190  ; 分流左_框架定點異常
3241  LDI     L4636  ; 進料分流左側旋轉定點ON
      ANI     L4646  ; 進料分流右側旋轉定點ON
      ANI     B24E  ; 進料分流旋臂變頻器INVA3運轉
      OUT     T4191 K10  ; 進料分流旋轉定點光電異常延遲
3248  LD      M4191  ; 分流_旋轉定點異常
      ANI     L4032  ; 爐體段  異常復歸
      OR      T4191  ; 進料分流旋轉定點光電異常延遲
      AND     T1000  ; 開機延遲
      OUT     M4191  ; 分流_旋轉定點異常
3253  LD      B8C  ; 分流右_框架上定點光電
      ANI     B8D  ; 分流右_框架下定點光電
      LDI     B8C  ; 分流右_框架上定點光電
      AND     B8D  ; 分流右_框架下定點光電
      ORB
      AND     L4642  ; 進料分流右側昇降上定點
      OUT     T4192 K10  ; 分流右_框架定點異常延遲
3263  LD      M4192  ; 分流右_框架定點異常
      ANI     L4032  ; 爐體段  異常復歸
      OR      T4192  ; 分流右_框架定點異常延遲
      AND     T1000  ; 開機延遲
      OUT     M4192  ; 分流右_框架定點異常
3268  LD      B92  ; 左IR輸送進框定位光纖
      AND     L4651  ; 左IR輸送進框補助上昇定點
      OUT     T4194 K5  ; 左IR進框補助光電異常延遲
3274  LD      M4194  ; 左側合流補助昇降框架光纖
      ANI     L4032  ; 爐體段  異常復歸
      OR      T4194  ; 左IR進框補助光電異常延遲
      AND     T1000  ; 開機延遲
      OUT     M4194  ; 左側合流補助昇降框架光纖
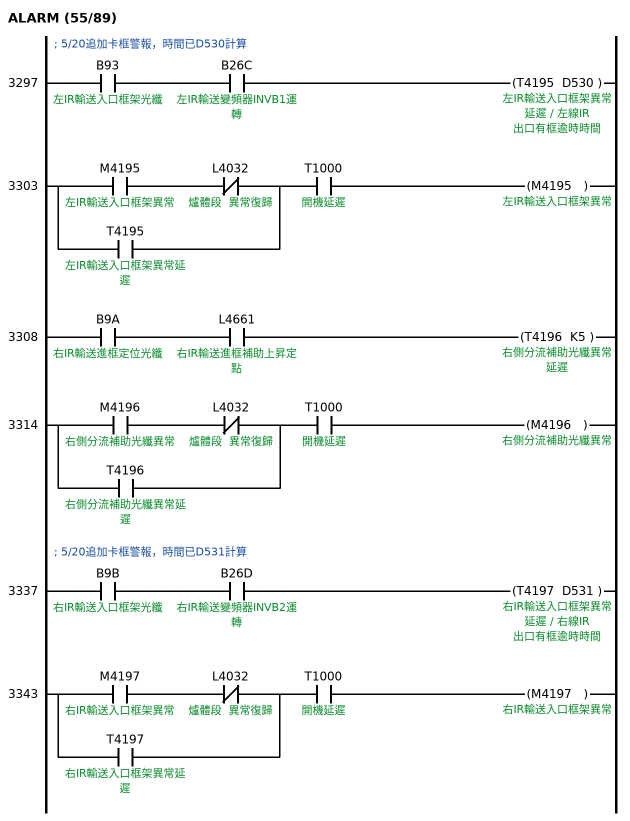
; 5/20追加卡框警報，時間已D530計算
3297  LD      B93  ; 左IR輸送入口框架光纖
      AND     B26C  ; 左IR輸送變頻器INVB1運轉
      OUT     T4195 D530  ; 左IR輸送入口框架異常延遲 / 左線IR  出口有框逾時時間
3303  LD      M4195  ; 左IR輸送入口框架異常
      ANI     L4032  ; 爐體段  異常復歸
      OR      T4195  ; 左IR輸送入口框架異常延遲
      AND     T1000  ; 開機延遲
      OUT     M4195  ; 左IR輸送入口框架異常
3308  LD      B9A  ; 右IR輸送進框定位光纖
      AND     L4661  ; 右IR輸送進框補助上昇定點
      OUT     T4196 K5  ; 右側分流補助光纖異常延遲
3314  LD      M4196  ; 右側分流補助光纖異常
      ANI     L4032  ; 爐體段  異常復歸
      OR      T4196  ; 右側分流補助光纖異常延遲
      AND     T1000  ; 開機延遲
      OUT     M4196  ; 右側分流補助光纖異常
; 5/20追加卡框警報，時間已D531計算
3337  LD      B9B  ; 右IR輸送入口框架光纖
      AND     B26D  ; 右IR輸送變頻器INVB2運轉
      OUT     T4197 D531  ; 右IR輸送入口框架異常延遲 / 右線IR  出口有框逾時時間
3343  LD      M4197  ; 右IR輸送入口框架異常
      ANI     L4032  ; 爐體段  異常復歸
      OR      T4197  ; 右IR輸送入口框架異常延遲
      AND     T1000  ; 開機延遲
      OUT     M4197  ; 右IR輸送入口框架異常
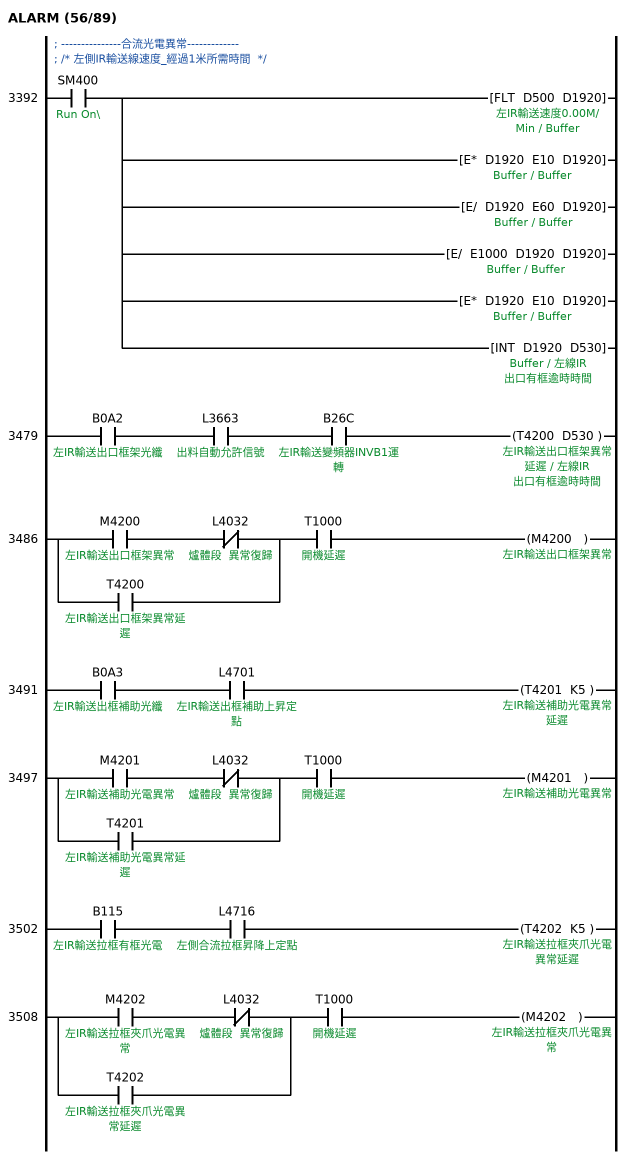
; ---------------合流光電異常-------------
; /* 左側IR輸送線速度_經過1米所需時間  */
3392  LD      SM400  ; Run On\
      FLT     D500 D1920  ; 左IR輸送速度0.00M/Min / Buffer
      E*      D1920 E10 D1920
        [note] /* 換算線速度單位_mm/M */
      E/      D1920 E60 D1920
        [note] /* 換算每秒移動距離_單位mm/S */
      E/      E1000 D1920 D1920
        [note] /* 計算每米需移動時間_Sec/M */
      E*      D1920 E10 D1920
        [note] /* 換算時間單位_0.1Sec */
      INT     D1920 D530
3479  LD      B0A2  ; 左IR輸送出口框架光纖
      AND     L3663  ; 出料自動允許信號
      AND     B26C  ; 左IR輸送變頻器INVB1運轉
      OUT     T4200 D530  ; 左IR輸送出口框架異常延遲 / 左線IR  出口有框逾時時間
3486  LD      M4200  ; 左IR輸送出口框架異常
      ANI     L4032  ; 爐體段  異常復歸
      OR      T4200  ; 左IR輸送出口框架異常延遲
      AND     T1000  ; 開機延遲
      OUT     M4200  ; 左IR輸送出口框架異常
3491  LD      B0A3  ; 左IR輸送出框補助光纖
      AND     L4701  ; 左IR輸送出框補助上昇定點
      OUT     T4201 K5  ; 左IR輸送補助光電異常延遲
3497  LD      M4201  ; 左IR輸送補助光電異常
      ANI     L4032  ; 爐體段  異常復歸
      OR      T4201  ; 左IR輸送補助光電異常延遲
      AND     T1000  ; 開機延遲
      OUT     M4201  ; 左IR輸送補助光電異常
3502  LD      B115  ; 左IR輸送拉框有框光電
      AND     L4716  ; 左側合流拉框昇降上定點
      OUT     T4202 K5  ; 左IR輸送拉框夾爪光電異常延遲
3508  LD      M4202  ; 左IR輸送拉框夾爪光電異常
      ANI     L4032  ; 爐體段  異常復歸
      OR      T4202  ; 左IR輸送拉框夾爪光電異常延遲
      AND     T1000  ; 開機延遲
      OUT     M4202  ; 左IR輸送拉框夾爪光電異常
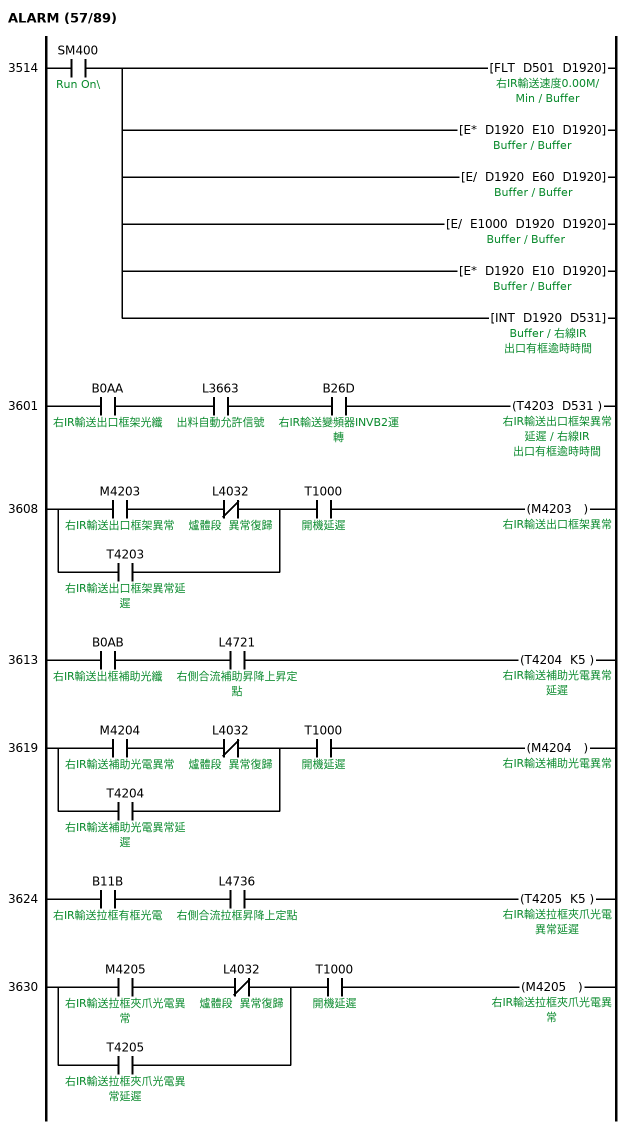
3514  LD      SM400  ; Run On\
      FLT     D501 D1920  ; 右IR輸送速度0.00M/Min
      E*      D1920 E10 D1920
        [note] /* 換算線速度單位_mm/M */
      E/      D1920 E60 D1920
        [note] /* 換算每秒移動距離_單位mm/S */
      E/      E1000 D1920 D1920
        [note] /* 計算每米需移動時間_Sec/M */
      E*      D1920 E10 D1920
        [note] /* 換算時間單位_0.1Sec */
      INT     D1920 D531
3601  LD      B0AA  ; 右IR輸送出口框架光纖
      AND     L3663  ; 出料自動允許信號
      AND     B26D  ; 右IR輸送變頻器INVB2運轉
      OUT     T4203 D531  ; 右IR輸送出口框架異常延遲 / 右線IR  出口有框逾時時間
3608  LD      M4203  ; 右IR輸送出口框架異常
      ANI     L4032  ; 爐體段  異常復歸
      OR      T4203  ; 右IR輸送出口框架異常延遲
      AND     T1000  ; 開機延遲
      OUT     M4203  ; 右IR輸送出口框架異常
3613  LD      B0AB  ; 右IR輸送出框補助光纖
      AND     L4721  ; 右側合流補助昇降上昇定點
      OUT     T4204 K5  ; 右IR輸送補助光電異常延遲
3619  LD      M4204  ; 右IR輸送補助光電異常
      ANI     L4032  ; 爐體段  異常復歸
      OR      T4204  ; 右IR輸送補助光電異常延遲
      AND     T1000  ; 開機延遲
      OUT     M4204  ; 右IR輸送補助光電異常
3624  LD      B11B  ; 右IR輸送拉框有框光電
      AND     L4736  ; 右側合流拉框昇降上定點
      OUT     T4205 K5  ; 右IR輸送拉框夾爪光電異常延遲
3630  LD      M4205  ; 右IR輸送拉框夾爪光電異常
      ANI     L4032  ; 爐體段  異常復歸
      OR      T4205  ; 右IR輸送拉框夾爪光電異常延遲
      AND     T1000  ; 開機延遲
      OUT     M4205  ; 右IR輸送拉框夾爪光電異常
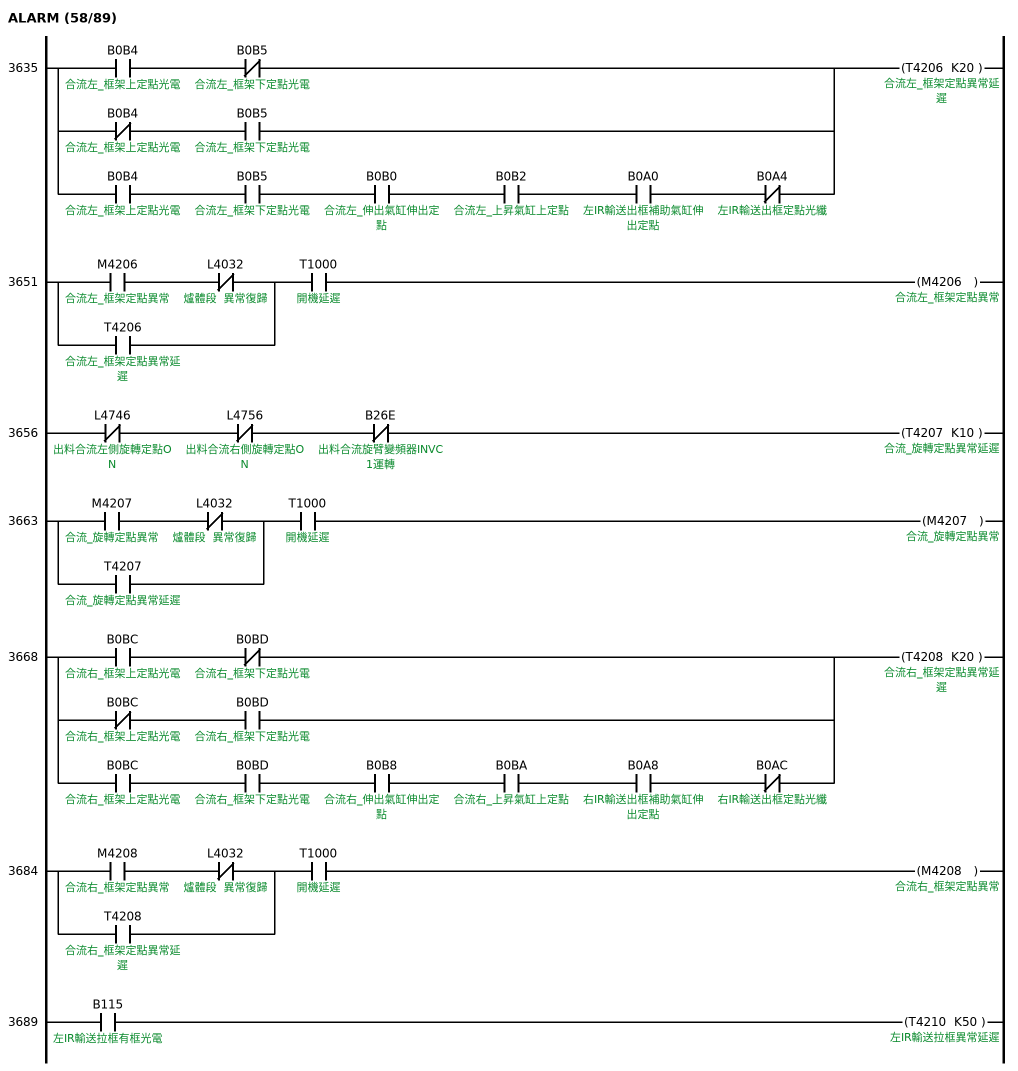
3635  LD      B0B4  ; 合流左_框架上定點光電
      ANI     B0B5  ; 合流左_框架下定點光電
      LDI     B0B4  ; 合流左_框架上定點光電
      AND     B0B5  ; 合流左_框架下定點光電
      ORB
      LD      B0B4  ; 合流左_框架上定點光電
      AND     B0B5  ; 合流左_框架下定點光電
      AND     B0B0  ; 合流左_伸出氣缸伸出定點
      AND     B0B2  ; 合流左_上昇氣缸上定點
      AND     B0A0  ; 左IR輸送出框補助氣缸伸出定點
      ANI     B0A4  ; 左IR輸送出框定點光纖
      ORB
      OUT     T4206 K20  ; 合流左_框架定點異常延遲
3651  LD      M4206  ; 合流左_框架定點異常
      ANI     L4032  ; 爐體段  異常復歸
      OR      T4206  ; 合流左_框架定點異常延遲
      AND     T1000  ; 開機延遲
      OUT     M4206  ; 合流左_框架定點異常
3656  LDI     L4746  ; 出料合流左側旋轉定點ON
      ANI     L4756  ; 出料合流右側旋轉定點ON
      ANI     B26E  ; 出料合流旋臂變頻器INVC1運轉
      OUT     T4207 K10  ; 合流_旋轉定點異常延遲
3663  LD      M4207  ; 合流_旋轉定點異常
      ANI     L4032  ; 爐體段  異常復歸
      OR      T4207  ; 合流_旋轉定點異常延遲
      AND     T1000  ; 開機延遲
      OUT     M4207  ; 合流_旋轉定點異常
3668  LD      B0BC  ; 合流右_框架上定點光電
      ANI     B0BD  ; 合流右_框架下定點光電
      LDI     B0BC  ; 合流右_框架上定點光電
      AND     B0BD  ; 合流右_框架下定點光電
      ORB
      LD      B0BC  ; 合流右_框架上定點光電
      AND     B0BD  ; 合流右_框架下定點光電
      AND     B0B8  ; 合流右_伸出氣缸伸出定點
      AND     B0BA  ; 合流右_上昇氣缸上定點
      AND     B0A8  ; 右IR輸送出框補助氣缸伸出定點
      ANI     B0AC  ; 右IR輸送出框定點光纖
      ORB
      OUT     T4208 K20  ; 合流右_框架定點異常延遲
3684  LD      M4208  ; 合流右_框架定點異常
      ANI     L4032  ; 爐體段  異常復歸
      OR      T4208  ; 合流右_框架定點異常延遲
      AND     T1000  ; 開機延遲
      OUT     M4208  ; 合流右_框架定點異常
3689  LD      B115  ; 左IR輸送拉框有框光電
      OUT     T4210 K50  ; 左IR輸送拉框異常延遲
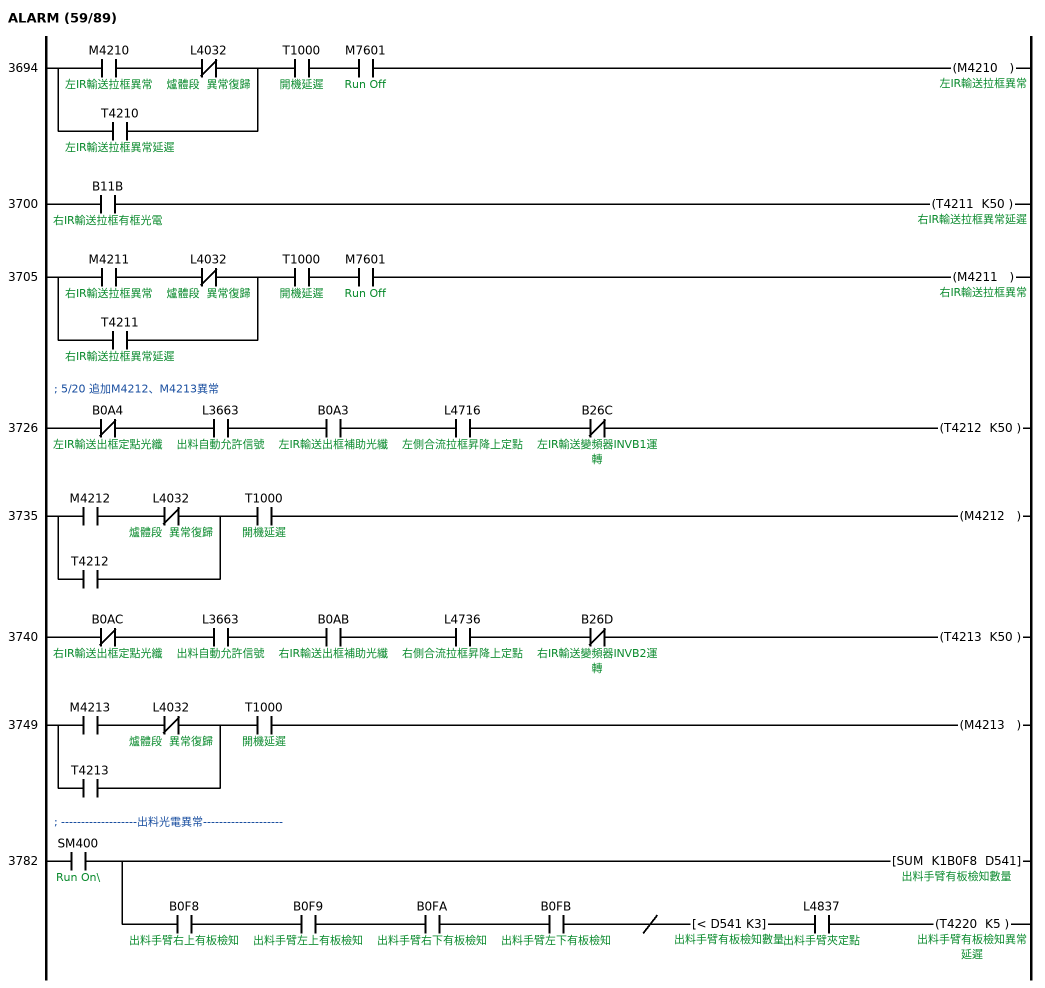
3694  LD      M4210  ; 左IR輸送拉框異常
      ANI     L4032  ; 爐體段  異常復歸
      OR      T4210  ; 左IR輸送拉框異常延遲
      AND     T1000  ; 開機延遲
      AND     M7601  ; Run Off
      OUT     M4210  ; 左IR輸送拉框異常
3700  LD      B11B  ; 右IR輸送拉框有框光電
      OUT     T4211 K50  ; 右IR輸送拉框異常延遲
3705  LD      M4211  ; 右IR輸送拉框異常
      ANI     L4032  ; 爐體段  異常復歸
      OR      T4211  ; 右IR輸送拉框異常延遲
      AND     T1000  ; 開機延遲
      AND     M7601  ; Run Off
      OUT     M4211  ; 右IR輸送拉框異常
; 5/20 追加M4212、M4213異常
3726  LDI     B0A4  ; 左IR輸送出框定點光纖
      AND     L3663  ; 出料自動允許信號
      AND     B0A3  ; 左IR輸送出框補助光纖
      AND     L4716  ; 左側合流拉框昇降上定點
      ANI     B26C  ; 左IR輸送變頻器INVB1運轉
      OUT     T4212 K50
3735  LD      M4212
      ANI     L4032  ; 爐體段  異常復歸
      OR      T4212
      AND     T1000  ; 開機延遲
      OUT     M4212
3740  LDI     B0AC  ; 右IR輸送出框定點光纖
      AND     L3663  ; 出料自動允許信號
      AND     B0AB  ; 右IR輸送出框補助光纖
      AND     L4736  ; 右側合流拉框昇降上定點
      ANI     B26D  ; 右IR輸送變頻器INVB2運轉
      OUT     T4213 K50
3749  LD      M4213
      ANI     L4032  ; 爐體段  異常復歸
      OR      T4213
      AND     T1000  ; 開機延遲
      OUT     M4213
; -------------------出料光電異常--------------------
3782  LD      SM400  ; Run On\
      SUM     K1B0F8 D541  ; 出料手臂右上有板檢知 / 出料手臂有板檢知數量
      AND     B0F8  ; 出料手臂右上有板檢知
      AND     B0F9  ; 出料手臂左上有板檢知
      AND     B0FA  ; 出料手臂右下有板檢知
      AND     B0FB  ; 出料手臂左下有板檢知
      INV
      AND<    D541 K3  ; 出料手臂有板檢知數量
      AND     L4837  ; 出料手臂夾定點
      OUT     T4220 K5  ; 出料手臂有板檢知異常延遲
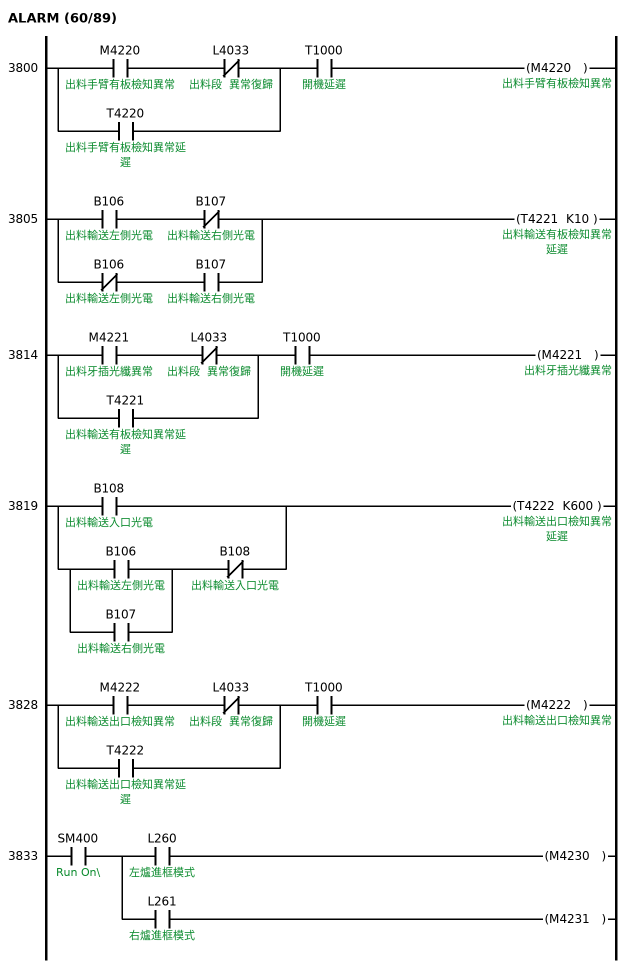
3800  LD      M4220  ; 出料手臂有板檢知異常
      ANI     L4033  ; 出料段  異常復歸
      OR      T4220  ; 出料手臂有板檢知異常延遲
      AND     T1000  ; 開機延遲
      OUT     M4220  ; 出料手臂有板檢知異常
3805  LD      B106  ; 出料輸送左側光電
      ANI     B107  ; 出料輸送右側光電
      LDI     B106  ; 出料輸送左側光電
      AND     B107  ; 出料輸送右側光電
      ORB
      OUT     T4221 K10  ; 出料輸送有板檢知異常延遲
3814  LD      M4221  ; 出料牙插光纖異常
      ANI     L4033  ; 出料段  異常復歸
      OR      T4221  ; 出料輸送有板檢知異常延遲
      AND     T1000  ; 開機延遲
      OUT     M4221  ; 出料牙插光纖異常
3819  LD      B108  ; 出料輸送入口光電
      LD      B106  ; 出料輸送左側光電
      OR      B107  ; 出料輸送右側光電
      ANI     B108  ; 出料輸送入口光電
      ORB
      OUT     T4222 K600  ; 出料輸送出口檢知異常延遲
3828  LD      M4222  ; 出料輸送出口檢知異常
      ANI     L4033  ; 出料段  異常復歸
      OR      T4222  ; 出料輸送出口檢知異常延遲
      AND     T1000  ; 開機延遲
      OUT     M4222  ; 出料輸送出口檢知異常
3833  LD      SM400  ; Run On\
      MPS
      AND     L260  ; 左爐進框模式
      OUT     M4230
      MPP
      AND     L261  ; 右爐進框模式
      OUT     M4231
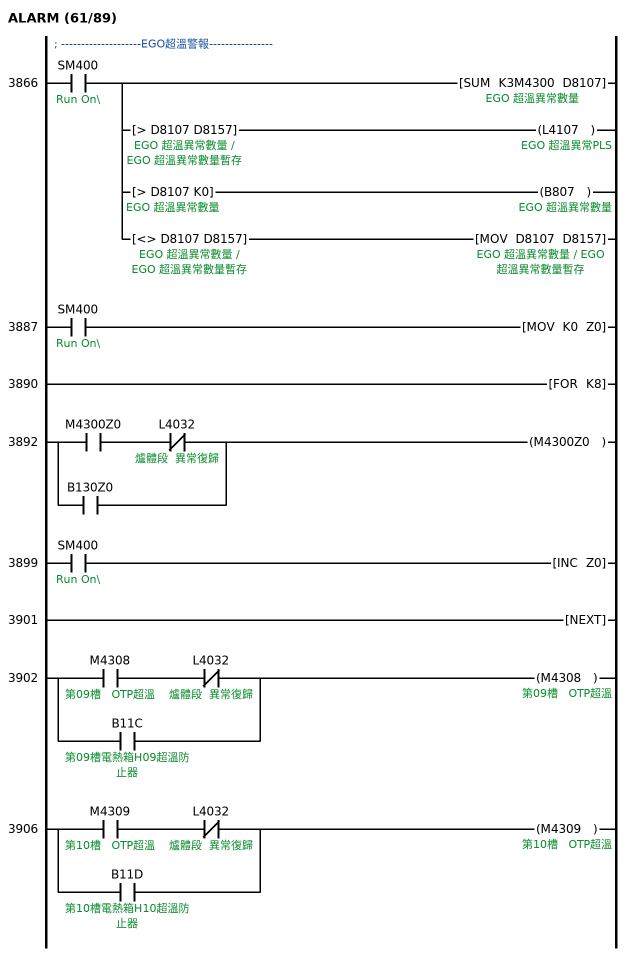
; --------------------EGO超溫警報----------------
3866  LD      SM400  ; Run On\
      SUM     K3M4300 D8107  ; 第01槽   OTP超溫 / EGO 超溫異常數量
      MPS
      AND>    D8107 D8157  ; EGO 超溫異常數量 / EGO 超溫異常數量暫存
      OUT     L4107  ; EGO 超溫異常PLS
      MRD
      AND>    D8107 K0  ; EGO 超溫異常數量
      OUT     B807  ; EGO 超溫異常數量
      MPP
      AND<>   D8107 D8157  ; EGO 超溫異常數量 / EGO 超溫異常數量暫存
      MOV     D8107 D8157
3887  LD      SM400  ; Run On\
      MOV     K0 Z0
3890  FOR     K8
3892  LD      M4300Z0
      ANI     L4032  ; 爐體段  異常復歸
      OR      B130Z0
      OUT     M4300Z0
3899  LD      SM400  ; Run On\
      INC     Z0
3901  NEXT
3902  LD      M4308  ; 第09槽   OTP超溫
      ANI     L4032  ; 爐體段  異常復歸
      OR      B11C  ; 第09槽電熱箱H09超溫防止器
      OUT     M4308  ; 第09槽   OTP超溫
3906  LD      M4309  ; 第10槽   OTP超溫
      ANI     L4032  ; 爐體段  異常復歸
      OR      B11D  ; 第10槽電熱箱H10超溫防止器
      OUT     M4309  ; 第10槽   OTP超溫
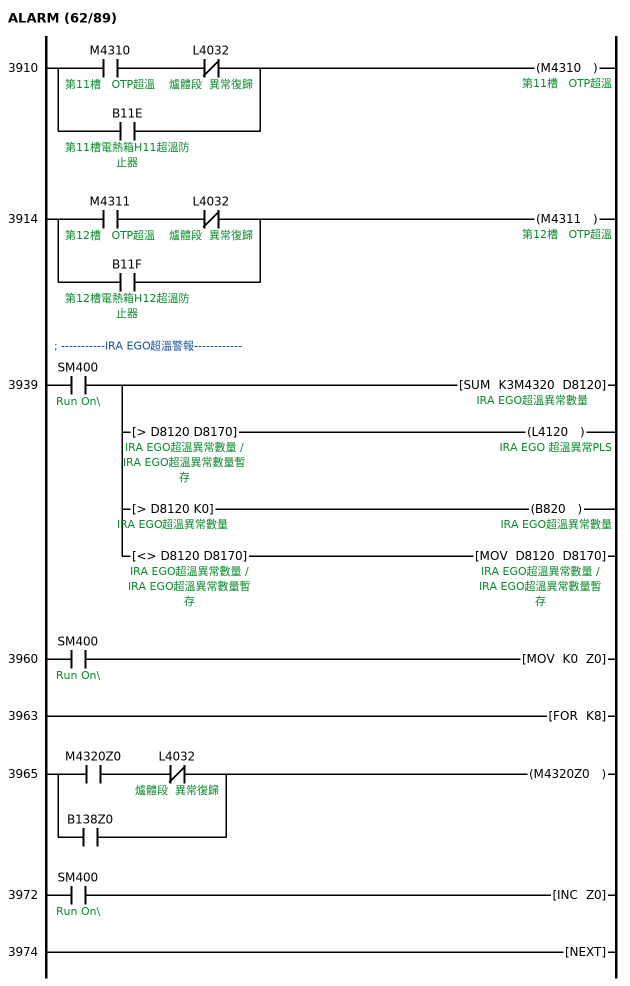
3910  LD      M4310  ; 第11槽   OTP超溫
      ANI     L4032  ; 爐體段  異常復歸
      OR      B11E  ; 第11槽電熱箱H11超溫防止器
      OUT     M4310  ; 第11槽   OTP超溫
3914  LD      M4311  ; 第12槽   OTP超溫
      ANI     L4032  ; 爐體段  異常復歸
      OR      B11F  ; 第12槽電熱箱H12超溫防止器
      OUT     M4311  ; 第12槽   OTP超溫
; -----------IRA EGO超溫警報------------
3939  LD      SM400  ; Run On\
      SUM     K3M4320 D8120  ; 第01槽  IRA OTP 超溫 / IRA EGO超溫異常數量
      MPS
      AND>    D8120 D8170  ; IRA EGO超溫異常數量 / IRA EGO超溫異常數量暫存
      OUT     L4120  ; IRA EGO 超溫異常PLS
      MRD
      AND>    D8120 K0  ; IRA EGO超溫異常數量
      OUT     B820  ; IRA EGO超溫異常數量
      MPP
      AND<>   D8120 D8170  ; IRA EGO超溫異常數量 / IRA EGO超溫異常數量暫存
      MOV     D8120 D8170
3960  LD      SM400  ; Run On\
      MOV     K0 Z0
3963  FOR     K8
3965  LD      M4320Z0
      ANI     L4032  ; 爐體段  異常復歸
      OR      B138Z0
      OUT     M4320Z0
3972  LD      SM400  ; Run On\
      INC     Z0
3974  NEXT
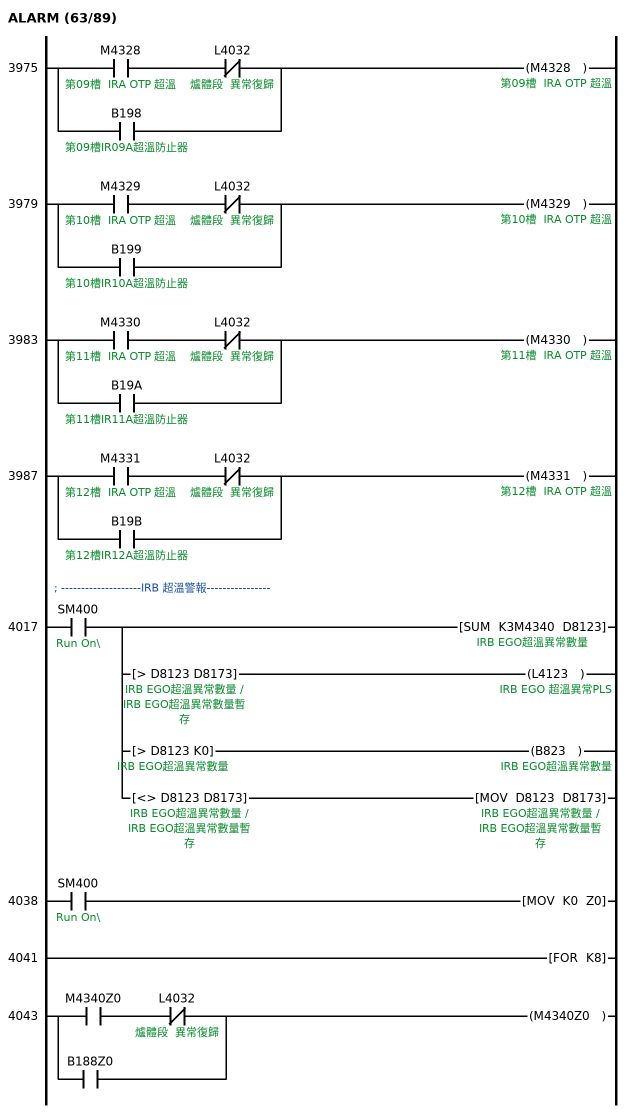
3975  LD      M4328  ; 第09槽  IRA OTP 超溫
      ANI     L4032  ; 爐體段  異常復歸
      OR      B198  ; 第09槽IR09A超溫防止器
      OUT     M4328  ; 第09槽  IRA OTP 超溫
3979  LD      M4329  ; 第10槽  IRA OTP 超溫
      ANI     L4032  ; 爐體段  異常復歸
      OR      B199  ; 第10槽IR10A超溫防止器
      OUT     M4329  ; 第10槽  IRA OTP 超溫
3983  LD      M4330  ; 第11槽  IRA OTP 超溫
      ANI     L4032  ; 爐體段  異常復歸
      OR      B19A  ; 第11槽IR11A超溫防止器
      OUT     M4330  ; 第11槽  IRA OTP 超溫
3987  LD      M4331  ; 第12槽  IRA OTP 超溫
      ANI     L4032  ; 爐體段  異常復歸
      OR      B19B  ; 第12槽IR12A超溫防止器
      OUT     M4331  ; 第12槽  IRA OTP 超溫
; --------------------IRB 超溫警報----------------
4017  LD      SM400  ; Run On\
      SUM     K3M4340 D8123  ; 第01槽  IRB OTP 超溫 / IRB EGO超溫異常數量
      MPS
      AND>    D8123 D8173  ; IRB EGO超溫異常數量 / IRB EGO超溫異常數量暫存
      OUT     L4123  ; IRB EGO 超溫異常PLS
      MRD
      AND>    D8123 K0  ; IRB EGO超溫異常數量
      OUT     B823  ; IRB EGO超溫異常數量
      MPP
      AND<>   D8123 D8173  ; IRB EGO超溫異常數量 / IRB EGO超溫異常數量暫存
      MOV     D8123 D8173
4038  LD      SM400  ; Run On\
      MOV     K0 Z0
4041  FOR     K8
4043  LD      M4340Z0
      ANI     L4032  ; 爐體段  異常復歸
      OR      B188Z0
      OUT     M4340Z0
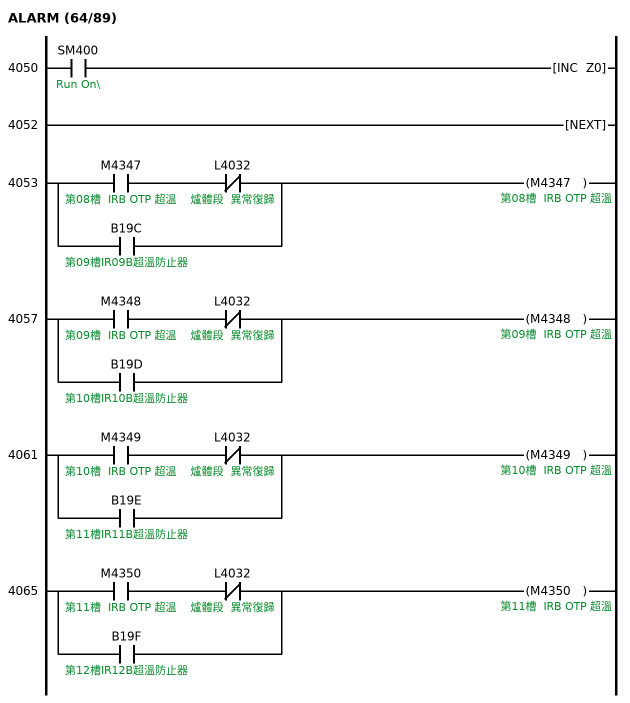
4050  LD      SM400  ; Run On\
      INC     Z0
4052  NEXT
4053  LD      M4347  ; 第08槽  IRB OTP 超溫
      ANI     L4032  ; 爐體段  異常復歸
      OR      B19C  ; 第09槽IR09B超溫防止器
      OUT     M4347  ; 第08槽  IRB OTP 超溫
4057  LD      M4348  ; 第09槽  IRB OTP 超溫
      ANI     L4032  ; 爐體段  異常復歸
      OR      B19D  ; 第10槽IR10B超溫防止器
      OUT     M4348  ; 第09槽  IRB OTP 超溫
4061  LD      M4349  ; 第10槽  IRB OTP 超溫
      ANI     L4032  ; 爐體段  異常復歸
      OR      B19E  ; 第11槽IR11B超溫防止器
      OUT     M4349  ; 第10槽  IRB OTP 超溫
4065  LD      M4350  ; 第11槽  IRB OTP 超溫
      ANI     L4032  ; 爐體段  異常復歸
      OR      B19F  ; 第12槽IR12B超溫防止器
      OUT     M4350  ; 第11槽  IRB OTP 超溫
